LIN {X 0,Y 682.383,Z 707.31,A -85,B 0,C 180,E1 4367.128,E2 4367.128} C_VEL
LIN {X 0,Y 682.576,Z 707.31,A -85,B 0,C 180,E1 4371.565,E2 4371.565} C_VEL
LIN {X 0,Y 682.448,Z 707.31,A -85,B 0,C 180,E1 4374.859,E2 4374.859} C_VEL
LIN {X 0,Y 694.724,Z 736.712,A -85,B 0,C 180,E1 4375.905,E2 4375.905} C_VEL
LIN {X 0,Y 693.686,Z 780.447,A -85,B 0,C 180,E1 4376.761,E2 4376.761} C_VEL
LIN {X 0,Y 692.089,Z 825.553,A -85,B 0,C 180,E1 4378.187,E2 4378.187} C_VEL
LIN {X 0,Y 690.132,Z 869.734,A -85,B 0,C 180,E1 4380.196,E2 4380.196} C_VEL
LIN {X 0,Y 688.071,Z 912.153,A -85,B 0,C 180,E1 4382.814,E2 4382.814} C_VEL
LIN {X 0,Y 686.387,Z 948.211,A -85,B 0,C 180,E1 4385.72,E2 4385.72} C_VEL
LIN {X 0,Y 684.951,Z 981.072,A -85,B 0,C 180,E1 4389.145,E2 4389.145} C_VEL
LIN {X 0,Y 684.052,Z 1007.657,A -85,B 0,C 180,E1 4392.773,E2 4392.773} C_VEL
LIN {X 0,Y 683.489,Z 1028.052,A -85,B 0,C 180,E1 4396.539,E2 4396.539} C_VEL
LIN {X 0,Y 683.179,Z 1041.813,A -85,B 0,C 180,E1 4400.192,E2 4400.192} C_VEL
LIN {X 0,Y 683.173,Z 1049.91,A -85,B 0,C 180,E1 4403.633,E2 4403.633} C_VEL
LIN {X 0,Y 683.009,Z 1053.376,A -85,B 0,C 180,E1 4407.457,E2 4407.457} C_VEL
LIN {X 0,Y 683.089,Z 1051.321,A -85,B 0,C 180,E1 4411.272,E2 4411.272} C_VEL
LIN {X 0,Y 683.176,Z 1045.315,A -85,B 0,C 180,E1 4414.453,E2 4414.453} C_VEL
LIN {X 0,Y 683.301,Z 1034.031,A -85,B 0,C 180,E1 4417.968,E2 4417.968} C_VEL
LIN {X 0,Y 683.712,Z 1015.525,A -85,B 0,C 180,E1 4421.831,E2 4421.831} C_VEL
LIN {X 0,Y 684.513,Z 990.501,A -85,B 0,C 180,E1 4425.594,E2 4425.594} C_VEL
LIN {X 0,Y 685.858,Z 958.739,A -85,B 0,C 180,E1 4429.188,E2 4429.188} C_VEL
LIN {X 0,Y 687.532,Z 923.074,A -85,B 0,C 180,E1 4432.291,E2 4432.291} C_VEL
LIN {X 0,Y 689.545,Z 882.981,A -85,B 0,C 180,E1 4434.973,E2 4434.973} C_VEL
LIN {X 0,Y 691.593,Z 838.894,A -85,B 0,C 180,E1 4437.183,E2 4437.183} C_VEL
LIN {X 0,Y 693.261,Z 795.202,A -85,B 0,C 180,E1 4438.745,E2 4438.745} C_VEL
LIN {X 0,Y 694.501,Z 752.579,A -85,B 0,C 180,E1 4439.746,E2 4439.746} C_VEL
LIN {X 0,Y 693.995,Z 732.964,A -85,B 0,C 180,E1 4440.096,E2 4440.096} C_VEL
LIN {X 0,Y 682.507,Z 707.31,A -85,B 0,C 180,E1 4441.104,E2 4441.104} C_VEL
LIN {X 0,Y 682.451,Z 707.31,A -85,B 0,C 180,E1 4446.925,E2 4446.925} C_VEL
LIN {X 0,Y 682.413,Z 707.31,A -85,B 0,C 180,E1 4451.775,E2 4451.775} C_VEL
LIN {X 0,Y 682.5,Z 707.31,A -85,B 0,C 180,E1 4457.116,E2 4457.116} C_VEL
LIN {X 0,Y 682.473,Z 707.31,A -85,B 0,C 180,E1 4461.555,E2 4461.555} C_VEL
LIN {X 0,Y 682.507,Z 707.31,A -85,B 0,C 180,E1 4466.281,E2 4466.281} C_VEL
LIN {X 0,Y 682.478,Z 707.31,A -85,B 0,C 180,E1 4470.756,E2 4470.756} C_VEL
LIN {X 0,Y 682.492,Z 707.31,A -85,B 0,C 180,E1 4475.557,E2 4475.557} C_VEL
LIN {X 0,Y 682.591,Z 707.31,A -85,B 0,C 180,E1 4480.546,E2 4480.546} C_VEL
LIN {X 0,Y 682.835,Z 707.31,A -85,B 0,C 180,E1 4485.868,E2 4485.868} C_VEL
LIN {X 0,Y 682.918,Z 707.31,A -85,B 0,C 180,E1 4491.062,E2 4491.062} C_VEL
LIN {X 0,Y 682.761,Z 707.31,A -85,B 0,C 180,E1 4496.18,E2 4496.18} C_VEL
LIN {X 0,Y 683.022,Z 707.31,A -85,B 0,C 180,E1 4501.269,E2 4501.269} C_VEL
LIN {X 0,Y 682.964,Z 707.31,A -85,B 0,C 180,E1 4507.648,E2 4507.648} C_VEL
LIN {X 0,Y 682.688,Z 707.31,A -85,B 0,C 180,E1 4512.823,E2 4512.823} C_VEL
LIN {X 0,Y 682.453,Z 707.31,A -85,B 0,C 180,E1 4518.109,E2 4518.109} C_VEL
LIN {X 0,Y 682.435,Z 707.31,A -85,B 0,C 180,E1 4521.572,E2 4521.572} C_VEL
LIN {X 0,Y 678.414,Z 707.31,A -85,B 0,C 180,E1 4523.005,E2 4523.005} C_VEL
LIN {X 0,Y 674.479,Z 707.31,A -85,B 0,C 180,E1 4524.456,E2 4524.456} C_VEL
LIN {X 0,Y 674.601,Z 707.31,A -85,B 0,C 180,E1 4529.614,E2 4529.614} C_VEL
LIN {X 0,Y 674.601,Z 707.31,A -85,B 0,C 180,E1 4534.163,E2 4534.163} C_VEL
LIN {X 0,Y 674.578,Z 707.31,A -85,B 0,C 180,E1 4538.973,E2 4538.973} C_VEL
LIN {X 0,Y 674.535,Z 707.31,A -85,B 0,C 180,E1 4544.138,E2 4544.138} C_VEL
LIN {X 0,Y 674.52,Z 707.31,A -85,B 0,C 180,E1 4549.801,E2 4549.801} C_VEL
LIN {X 0,Y 674.478,Z 707.31,A -85,B 0,C 180,E1 4554.256,E2 4554.256} C_VEL
LIN {X 0,Y 674.508,Z 708.066,A -85,B 0,C 180,E1 4556.111,E2 4556.111} C_VEL
LIN {X 0,Y 688.176,Z 737.551,A -85,B 0,C 180,E1 4557.231,E2 4557.231} C_VEL
LIN {X 0,Y 687.447,Z 791.806,A -85,B 0,C 180,E1 4558.03,E2 4558.03} C_VEL
LIN {X 0,Y 685.87,Z 838.816,A -85,B 0,C 180,E1 4559.294,E2 4559.294} C_VEL
LIN {X 0,Y 683.746,Z 884.753,A -85,B 0,C 180,E1 4561.162,E2 4561.162} C_VEL
LIN {X 0,Y 681.479,Z 927.902,A -85,B 0,C 180,E1 4563.593,E2 4563.593} C_VEL
LIN {X 0,Y 679.459,Z 966.912,A -85,B 0,C 180,E1 4566.505,E2 4566.505} C_VEL
LIN {X 0,Y 677.682,Z 1000.895,A -85,B 0,C 180,E1 4569.793,E2 4569.793} C_VEL
LIN {X 0,Y 676.498,Z 1029.549,A -85,B 0,C 180,E1 4573.404,E2 4573.404} C_VEL
LIN {X 0,Y 675.771,Z 1053.159,A -85,B 0,C 180,E1 4577.409,E2 4577.409} C_VEL
LIN {X 0,Y 675.4,Z 1069.16,A -85,B 0,C 180,E1 4581.288,E2 4581.288} C_VEL
LIN {X 0,Y 675.235,Z 1078.459,A -85,B 0,C 180,E1 4584.849,E2 4584.849} C_VEL
LIN {X 0,Y 675.177,Z 1083.168,A -85,B 0,C 180,E1 4588.713,E2 4588.713} C_VEL
LIN {X 0,Y 675.3,Z 1082.218,A -85,B 0,C 180,E1 4592.572,E2 4592.572} C_VEL
LIN {X 0,Y 675.237,Z 1075.636,A -85,B 0,C 180,E1 4596.442,E2 4596.442} C_VEL
LIN {X 0,Y 675.368,Z 1064.65,A -85,B 0,C 180,E1 4599.981,E2 4599.981} C_VEL
LIN {X 0,Y 675.764,Z 1047.785,A -85,B 0,C 180,E1 4603.618,E2 4603.618} C_VEL
LIN {X 0,Y 676.601,Z 1025.27,A -85,B 0,C 180,E1 4607.192,E2 4607.192} C_VEL
LIN {X 0,Y 677.818,Z 997.464,A -85,B 0,C 180,E1 4610.573,E2 4610.573} C_VEL
LIN {X 0,Y 679.494,Z 964.868,A -85,B 0,C 180,E1 4613.667,E2 4613.667} C_VEL
LIN {X 0,Y 681.608,Z 926.092,A -85,B 0,C 180,E1 4616.52,E2 4616.52} C_VEL
LIN {X 0,Y 683.832,Z 883.698,A -85,B 0,C 180,E1 4618.886,E2 4618.886} C_VEL
LIN {X 0,Y 685.911,Z 837.811,A -85,B 0,C 180,E1 4620.74,E2 4620.74} C_VEL
LIN {X 0,Y 687.491,Z 790.369,A -85,B 0,C 180,E1 4622.002,E2 4622.002} C_VEL
LIN {X 0,Y 687.505,Z 735.67,A -85,B 0,C 180,E1 4622.828,E2 4622.828} C_VEL
LIN {X 0,Y 674.593,Z 707.31,A -85,B 0,C 180,E1 4623.954,E2 4623.954} C_VEL
LIN {X 0,Y 674.584,Z 707.31,A -85,B 0,C 180,E1 4628.975,E2 4628.975} C_VEL
LIN {X 0,Y 674.547,Z 707.31,A -85,B 0,C 180,E1 4634.14,E2 4634.14} C_VEL
LIN {X 0,Y 674.52,Z 707.31,A -85,B 0,C 180,E1 4639.804,E2 4639.804} C_VEL
LIN {X 0,Y 674.531,Z 707.31,A -85,B 0,C 180,E1 4644.263,E2 4644.263} C_VEL
LIN {X 0,Y 674.635,Z 707.31,A -85,B 0,C 180,E1 4648.896,E2 4648.896} C_VEL
LIN {X 0,Y 674.568,Z 707.31,A -85,B 0,C 180,E1 4654.736,E2 4654.736} C_VEL
LIN {X 0,Y 674.678,Z 707.31,A -85,B 0,C 180,E1 4660.623,E2 4660.623} C_VEL
LIN {X 0,Y 674.746,Z 707.31,A -85,B 0,C 180,E1 4665.7,E2 4665.7} C_VEL
LIN {X 0,Y 674.975,Z 707.31,A -85,B 0,C 180,E1 4671.056,E2 4671.056} C_VEL
LIN {X 0,Y 674.685,Z 707.31,A -85,B 0,C 180,E1 4674.848,E2 4674.848} C_VEL
LIN {X 0,Y 674.832,Z 707.31,A -85,B 0,C 180,E1 4680.002,E2 4680.002} C_VEL
LIN {X 0,Y 674.973,Z 707.31,A -85,B 0,C 180,E1 4685.155,E2 4685.155} C_VEL
LIN {X 0,Y 674.842,Z 707.31,A -85,B 0,C 180,E1 4691.662,E2 4691.662} C_VEL
LIN {X 0,Y 674.512,Z 707.31,A -85,B 0,C 180,E1 4696.984,E2 4696.984} C_VEL
LIN {X 0,Y 674.815,Z 707.31,A -85,B 0,C 180,E1 4701.06,E2 4701.06} C_VEL
LIN {X 0,Y 674.524,Z 707.31,A -85,B 0,C 180,E1 4706.021,E2 4706.021} C_VEL
LIN {X 0,Y 674.373,Z 707.31,A -85,B 0,C 180,E1 4711.362,E2 4711.362} C_VEL
LIN {X 0,Y 674.46,Z 707.31,A -85,B 0,C 180,E1 4716.016,E2 4716.016} C_VEL
LIN {X 0,Y 674.591,Z 707.31,A -85,B 0,C 180,E1 4720.654,E2 4720.654} C_VEL
LIN {X 0,Y 674.533,Z 707.31,A -85,B 0,C 180,E1 4725.967,E2 4725.967} C_VEL
LIN {X 0,Y 674.655,Z 707.31,A -85,B 0,C 180,E1 4731.831,E2 4731.831} C_VEL
LIN {X 0,Y 674.543,Z 707.726,A -85,B 0,C 180,E1 4734.439,E2 4734.439} C_VEL
LIN {X 0,Y 688.006,Z 738.757,A -85,B 0,C 180,E1 4735.584,E2 4735.584} C_VEL
LIN {X 0,Y 686.802,Z 782.385,A -85,B 0,C 180,E1 4736.467,E2 4736.467} C_VEL
LIN {X 0,Y 685.108,Z 826.206,A -85,B 0,C 180,E1 4737.881,E2 4737.881} C_VEL
LIN {X 0,Y 682.962,Z 870.549,A -85,B 0,C 180,E1 4739.927,E2 4739.927} C_VEL
LIN {X 0,Y 680.722,Z 912.029,A -85,B 0,C 180,E1 4742.514,E2 4742.514} C_VEL
LIN {X 0,Y 678.777,Z 949.734,A -85,B 0,C 180,E1 4745.606,E2 4745.606} C_VEL
LIN {X 0,Y 677.211,Z 981.864,A -85,B 0,C 180,E1 4749.021,E2 4749.021} C_VEL
LIN {X 0,Y 676.257,Z 1007.816,A -85,B 0,C 180,E1 4752.619,E2 4752.619} C_VEL
LIN {X 0,Y 675.644,Z 1027.935,A -85,B 0,C 180,E1 4756.379,E2 4756.379} C_VEL
LIN {X 0,Y 675.323,Z 1041.566,A -85,B 0,C 180,E1 4760.018,E2 4760.018} C_VEL
LIN {X 0,Y 675.273,Z 1049.865,A -85,B 0,C 180,E1 4763.558,E2 4763.558} C_VEL
LIN {X 0,Y 675.125,Z 1053.369,A -85,B 0,C 180,E1 4767.428,E2 4767.428} C_VEL
LIN {X 0,Y 675.205,Z 1051.353,A -85,B 0,C 180,E1 4771.287,E2 4771.287} C_VEL
LIN {X 0,Y 675.249,Z 1043.77,A -85,B 0,C 180,E1 4775.151,E2 4775.151} C_VEL
LIN {X 0,Y 675.418,Z 1031.467,A -85,B 0,C 180,E1 4778.711,E2 4778.711} C_VEL
LIN {X 0,Y 675.912,Z 1014.099,A -85,B 0,C 180,E1 4782.237,E2 4782.237} C_VEL
LIN {X 0,Y 676.833,Z 989.858,A -85,B 0,C 180,E1 4785.886,E2 4785.886} C_VEL
LIN {X 0,Y 678.252,Z 959.002,A -85,B 0,C 180,E1 4789.412,E2 4789.412} C_VEL
LIN {X 0,Y 680.132,Z 922.968,A -85,B 0,C 180,E1 4792.581,E2 4792.581} C_VEL
LIN {X 0,Y 682.333,Z 883.236,A -85,B 0,C 180,E1 4795.267,E2 4795.267} C_VEL
LIN {X 0,Y 684.626,Z 838.791,A -85,B 0,C 180,E1 4797.514,E2 4797.514} C_VEL
LIN {X 0,Y 686.388,Z 796.028,A -85,B 0,C 180,E1 4799.06,E2 4799.06} C_VEL
LIN {X 0,Y 687.752,Z 754.022,A -85,B 0,C 180,E1 4800.068,E2 4800.068} C_VEL
LIN {X 0,Y 687.42,Z 735.913,A -85,B 0,C 180,E1 4800.398,E2 4800.398} C_VEL
LIN {X 0,Y 674.524,Z 707.31,A -85,B 0,C 180,E1 4801.552,E2 4801.552} C_VEL
LIN {X 0,Y 674.521,Z 707.31,A -85,B 0,C 180,E1 4807.344,E2 4807.344} C_VEL
LIN {X 0,Y 674.469,Z 707.31,A -85,B 0,C 180,E1 4812.38,E2 4812.38} C_VEL
LIN {X 0,Y 674.605,Z 707.31,A -85,B 0,C 180,E1 4817.843,E2 4817.843} C_VEL
LIN {X 0,Y 674.527,Z 707.31,A -85,B 0,C 180,E1 4822.655,E2 4822.655} C_VEL
LIN {X 0,Y 674.622,Z 707.31,A -85,B 0,C 180,E1 4827.375,E2 4827.375} C_VEL
LIN {X 0,Y 674.57,Z 707.31,A -85,B 0,C 180,E1 4831.849,E2 4831.849} C_VEL
LIN {X 0,Y 674.476,Z 707.31,A -85,B 0,C 180,E1 4837.101,E2 4837.101} C_VEL
LIN {X 0,Y 674.536,Z 707.31,A -85,B 0,C 180,E1 4841.666,E2 4841.666} C_VEL
LIN {X 0,Y 675.041,Z 707.31,A -85,B 0,C 180,E1 4847.025,E2 4847.025} C_VEL
LIN {X 0,Y 674.947,Z 707.31,A -85,B 0,C 180,E1 4852.256,E2 4852.256} C_VEL
LIN {X 0,Y 674.865,Z 707.31,A -85,B 0,C 180,E1 4856.135,E2 4856.135} C_VEL
LIN {X 0,Y 675.128,Z 707.31,A -85,B 0,C 180,E1 4861.284,E2 4861.284} C_VEL
LIN {X 0,Y 675.046,Z 707.31,A -85,B 0,C 180,E1 4867.738,E2 4867.738} C_VEL
LIN {X 0,Y 674.77,Z 707.31,A -85,B 0,C 180,E1 4872.976,E2 4872.976} C_VEL
LIN {X 0,Y 674.551,Z 707.31,A -85,B 0,C 180,E1 4878.329,E2 4878.329} C_VEL
LIN {X 0,Y 674.451,Z 707.31,A -85,B 0,C 180,E1 4882.894,E2 4882.894} C_VEL
LIN {X 0,Y 674.479,Z 707.31,A -85,B 0,C 180,E1 4884.456,E2 4884.456} C_VEL
LIN {X 0,Y 670.595,Z 707.31,A -85,B 0,C 180,E1 4885.904,E2 4885.904} C_VEL
LIN {X 0,Y 666.66,Z 707.31,A -85,B 0,C 180,E1 4887.369,E2 4887.369} C_VEL
LIN {X 0,Y 666.712,Z 707.31,A -85,B 0,C 180,E1 4893.056,E2 4893.056} C_VEL
LIN {X 0,Y 666.637,Z 707.31,A -85,B 0,C 180,E1 4897.859,E2 4897.859} C_VEL
LIN {X 0,Y 666.548,Z 707.31,A -85,B 0,C 180,E1 4903.32,E2 4903.32} C_VEL
LIN {X 0,Y 666.538,Z 707.31,A -85,B 0,C 180,E1 4908.751,E2 4908.751} C_VEL
LIN {X 0,Y 666.576,Z 707.31,A -85,B 0,C 180,E1 4913.765,E2 4913.765} C_VEL
LIN {X 0,Y 666.565,Z 707.31,A -85,B 0,C 180,E1 4915.64,E2 4915.64} C_VEL
LIN {X 0,Y 681.528,Z 740.134,A -85,B 0,C 180,E1 4916.902,E2 4916.902} C_VEL
LIN {X 0,Y 680.677,Z 792.992,A -85,B 0,C 180,E1 4917.702,E2 4917.702} C_VEL
LIN {X 0,Y 678.976,Z 839.749,A -85,B 0,C 180,E1 4918.984,E2 4918.984} C_VEL
LIN {X 0,Y 676.703,Z 884.982,A -85,B 0,C 180,E1 4920.845,E2 4920.845} C_VEL
LIN {X 0,Y 674.264,Z 927.901,A -85,B 0,C 180,E1 4923.288,E2 4923.288} C_VEL
LIN {X 0,Y 671.967,Z 966.911,A -85,B 0,C 180,E1 4926.227,E2 4926.227} C_VEL
LIN {X 0,Y 670.1,Z 1000.051,A -85,B 0,C 180,E1 4929.459,E2 4929.459} C_VEL
LIN {X 0,Y 668.709,Z 1029.55,A -85,B 0,C 180,E1 4933.205,E2 4933.205} C_VEL
LIN {X 0,Y 667.954,Z 1052.672,A -85,B 0,C 180,E1 4937.157,E2 4937.157} C_VEL
LIN {X 0,Y 667.533,Z 1069.16,A -85,B 0,C 180,E1 4941.185,E2 4941.185} C_VEL
LIN {X 0,Y 667.352,Z 1078.459,A -85,B 0,C 180,E1 4944.788,E2 4944.788} C_VEL
LIN {X 0,Y 667.278,Z 1083.167,A -85,B 0,C 180,E1 4948.698,E2 4948.698} C_VEL
LIN {X 0,Y 667.428,Z 1082.217,A -85,B 0,C 180,E1 4952.602,E2 4952.602} C_VEL
LIN {X 0,Y 667.344,Z 1075.636,A -85,B 0,C 180,E1 4956.519,E2 4956.519} C_VEL
LIN {X 0,Y 667.512,Z 1064.516,A -85,B 0,C 180,E1 4960.133,E2 4960.133} C_VEL
LIN {X 0,Y 668.06,Z 1046.033,A -85,B 0,C 180,E1 4964.113,E2 4964.113} C_VEL
LIN {X 0,Y 669.136,Z 1021.013,A -85,B 0,C 180,E1 4967.987,E2 4967.987} C_VEL
LIN {X 0,Y 670.698,Z 989.205,A -85,B 0,C 180,E1 4971.691,E2 4971.691} C_VEL
LIN {X 0,Y 672.742,Z 953.245,A -85,B 0,C 180,E1 4974.894,E2 4974.894} C_VEL
LIN {X 0,Y 675.122,Z 912.935,A -85,B 0,C 180,E1 4977.647,E2 4977.647} C_VEL
LIN {X 0,Y 677.594,Z 868.414,A -85,B 0,C 180,E1 4979.913,E2 4979.913} C_VEL
LIN {X 0,Y 679.642,Z 822.708,A -85,B 0,C 180,E1 4981.559,E2 4981.559} C_VEL
LIN {X 0,Y 681.145,Z 773.641,A -85,B 0,C 180,E1 4982.662,E2 4982.662} C_VEL
LIN {X 0,Y 680.831,Z 737.977,A -85,B 0,C 180,E1 4983.163,E2 4983.163} C_VEL
LIN {X 0,Y 666.664,Z 707.31,A -85,B 0,C 180,E1 4984.388,E2 4984.388} C_VEL
LIN {X 0,Y 666.651,Z 707.31,A -85,B 0,C 180,E1 4989.529,E2 4989.529} C_VEL
LIN {X 0,Y 666.561,Z 707.31,A -85,B 0,C 180,E1 4995.193,E2 4995.193} C_VEL
LIN {X 0,Y 666.634,Z 707.31,A -85,B 0,C 180,E1 5000.613,E2 5000.613} C_VEL
LIN {X 0,Y 666.621,Z 707.31,A -85,B 0,C 180,E1 5005.371,E2 5005.371} C_VEL
LIN {X 0,Y 666.665,Z 707.31,A -85,B 0,C 180,E1 5009.998,E2 5009.998} C_VEL
LIN {X 0,Y 666.584,Z 707.31,A -85,B 0,C 180,E1 5015.414,E2 5015.414} C_VEL
LIN {X 0,Y 666.727,Z 707.31,A -85,B 0,C 180,E1 5020.069,E2 5020.069} C_VEL
LIN {X 0,Y 666.82,Z 707.31,A -85,B 0,C 180,E1 5025.526,E2 5025.526} C_VEL
LIN {X 0,Y 667.069,Z 707.31,A -85,B 0,C 180,E1 5030.852,E2 5030.852} C_VEL
LIN {X 0,Y 666.809,Z 707.31,A -85,B 0,C 180,E1 5034.787,E2 5034.787} C_VEL
LIN {X 0,Y 666.943,Z 707.31,A -85,B 0,C 180,E1 5040.002,E2 5040.002} C_VEL
LIN {X 0,Y 667.051,Z 707.31,A -85,B 0,C 180,E1 5045.216,E2 5045.216} C_VEL
LIN {X 0,Y 666.911,Z 707.31,A -85,B 0,C 180,E1 5051.803,E2 5051.803} C_VEL
LIN {X 0,Y 666.589,Z 707.31,A -85,B 0,C 180,E1 5057.292,E2 5057.292} C_VEL
LIN {X 0,Y 666.887,Z 707.31,A -85,B 0,C 180,E1 5061.322,E2 5061.322} C_VEL
LIN {X 0,Y 666.657,Z 707.31,A -85,B 0,C 180,E1 5065.59,E2 5065.59} C_VEL
LIN {X 0,Y 666.486,Z 707.31,A -85,B 0,C 180,E1 5070.231,E2 5070.231} C_VEL
LIN {X 0,Y 666.516,Z 707.31,A -85,B 0,C 180,E1 5075.066,E2 5075.066} C_VEL
LIN {X 0,Y 666.674,Z 707.31,A -85,B 0,C 180,E1 5079.531,E2 5079.531} C_VEL
LIN {X 0,Y 666.582,Z 707.31,A -85,B 0,C 180,E1 5085.192,E2 5085.192} C_VEL
LIN {X 0,Y 666.718,Z 707.31,A -85,B 0,C 180,E1 5090.608,E2 5090.608} C_VEL
LIN {X 0,Y 666.656,Z 707.711,A -85,B 0,C 180,E1 5093.986,E2 5093.986} C_VEL
LIN {X 0,Y 681.297,Z 740.305,A -85,B 0,C 180,E1 5095.248,E2 5095.248} C_VEL
LIN {X 0,Y 679.935,Z 785.032,A -85,B 0,C 180,E1 5096.188,E2 5096.188} C_VEL
LIN {X 0,Y 678.07,Z 828.293,A -85,B 0,C 180,E1 5097.627,E2 5097.627} C_VEL
LIN {X 0,Y 675.759,Z 871.521,A -85,B 0,C 180,E1 5099.659,E2 5099.659} C_VEL
LIN {X 0,Y 673.373,Z 912.455,A -85,B 0,C 180,E1 5102.25,E2 5102.25} C_VEL
LIN {X 0,Y 671.228,Z 949.46,A -85,B 0,C 180,E1 5105.313,E2 5105.313} C_VEL
LIN {X 0,Y 669.5,Z 981.657,A -85,B 0,C 180,E1 5108.768,E2 5108.768} C_VEL
LIN {X 0,Y 668.432,Z 1008.425,A -85,B 0,C 180,E1 5112.537,E2 5112.537} C_VEL
LIN {X 0,Y 667.727,Z 1029.34,A -85,B 0,C 180,E1 5116.549,E2 5116.549} C_VEL
LIN {X 0,Y 667.406,Z 1042.365,A -85,B 0,C 180,E1 5120.196,E2 5120.196} C_VEL
LIN {X 0,Y 667.373,Z 1049.821,A -85,B 0,C 180,E1 5123.482,E2 5123.482} C_VEL
LIN {X 0,Y 667.228,Z 1053.363,A -85,B 0,C 180,E1 5127.397,E2 5127.397} C_VEL
LIN {X 0,Y 667.304,Z 1051.385,A -85,B 0,C 180,E1 5131.302,E2 5131.302} C_VEL
LIN {X 0,Y 667.367,Z 1043.842,A -85,B 0,C 180,E1 5135.212,E2 5135.212} C_VEL
LIN {X 0,Y 667.552,Z 1031.573,A -85,B 0,C 180,E1 5138.814,E2 5138.814} C_VEL
LIN {X 0,Y 668.097,Z 1013.892,A -85,B 0,C 180,E1 5142.443,E2 5142.443} C_VEL
LIN {X 0,Y 669.101,Z 989.793,A -85,B 0,C 180,E1 5146.108,E2 5146.108} C_VEL
LIN {X 0,Y 670.644,Z 959.267,A -85,B 0,C 180,E1 5149.641,E2 5149.641} C_VEL
LIN {X 0,Y 672.762,Z 923.021,A -85,B 0,C 180,E1 5152.865,E2 5152.865} C_VEL
LIN {X 0,Y 675.23,Z 882.54,A -85,B 0,C 180,E1 5155.621,E2 5155.621} C_VEL
LIN {X 0,Y 677.681,Z 838.342,A -85,B 0,C 180,E1 5157.867,E2 5157.867} C_VEL
LIN {X 0,Y 679.638,Z 794.078,A -85,B 0,C 180,E1 5159.469,E2 5159.469} C_VEL
LIN {X 0,Y 681.118,Z 751.141,A -85,B 0,C 180,E1 5160.474,E2 5160.474} C_VEL
LIN {X 0,Y 680.665,Z 738.196,A -85,B 0,C 180,E1 5160.727,E2 5160.727} C_VEL
LIN {X 0,Y 666.588,Z 707.31,A -85,B 0,C 180,E1 5161.955,E2 5161.955} C_VEL
LIN {X 0,Y 666.639,Z 707.31,A -85,B 0,C 180,E1 5167.863,E2 5167.863} C_VEL
LIN {X 0,Y 666.541,Z 707.31,A -85,B 0,C 180,E1 5173.318,E2 5173.318} C_VEL
LIN {X 0,Y 666.647,Z 707.31,A -85,B 0,C 180,E1 5178.757,E2 5178.757} C_VEL
LIN {X 0,Y 666.62,Z 707.31,A -85,B 0,C 180,E1 5183.766,E2 5183.766} C_VEL
LIN {X 0,Y 666.726,Z 707.31,A -85,B 0,C 180,E1 5188.48,E2 5188.48} C_VEL
LIN {X 0,Y 666.702,Z 707.31,A -85,B 0,C 180,E1 5194.412,E2 5194.412} C_VEL
LIN {X 0,Y 666.74,Z 707.31,A -85,B 0,C 180,E1 5200.064,E2 5200.064} C_VEL
LIN {X 0,Y 666.936,Z 707.31,A -85,B 0,C 180,E1 5205.524,E2 5205.524} C_VEL
LIN {X 0,Y 667.092,Z 707.31,A -85,B 0,C 180,E1 5210.848,E2 5210.848} C_VEL
LIN {X 0,Y 666.985,Z 707.31,A -85,B 0,C 180,E1 5216.089,E2 5216.089} C_VEL
LIN {X 0,Y 667.058,Z 707.31,A -85,B 0,C 180,E1 5221.648,E2 5221.648} C_VEL
LIN {X 0,Y 667.131,Z 707.31,A -85,B 0,C 180,E1 5227.831,E2 5227.831} C_VEL
LIN {X 0,Y 666.862,Z 707.31,A -85,B 0,C 180,E1 5233.132,E2 5233.132} C_VEL
LIN {X 0,Y 666.661,Z 707.31,A -85,B 0,C 180,E1 5238.554,E2 5238.554} C_VEL
LIN {X 0,Y 666.562,Z 707.31,A -85,B 0,C 180,E1 5242.733,E2 5242.733} C_VEL
LIN {X 0,Y 666.66,Z 707.31,A -85,B 0,C 180,E1 5247.369,E2 5247.369} C_VEL
LIN {X 0,Y 662.663,Z 707.31,A -85,B 0,C 180,E1 5248.838,E2 5248.838} C_VEL
LIN {X 0,Y 658.79,Z 707.31,A -85,B 0,C 180,E1 5250.325,E2 5250.325} C_VEL
LIN {X 0,Y 658.748,Z 707.31,A -85,B 0,C 180,E1 5255.104,E2 5255.104} C_VEL
LIN {X 0,Y 658.617,Z 707.31,A -85,B 0,C 180,E1 5260.597,E2 5260.597} C_VEL
LIN {X 0,Y 658.605,Z 707.31,A -85,B 0,C 180,E1 5266.347,E2 5266.347} C_VEL
LIN {X 0,Y 658.665,Z 707.31,A -85,B 0,C 180,E1 5271.596,E2 5271.596} C_VEL
LIN {X 0,Y 658.652,Z 707.31,A -85,B 0,C 180,E1 5275.154,E2 5275.154} C_VEL
LIN {X 0,Y 674.979,Z 744.406,A -85,B 0,C 180,E1 5276.592,E2 5276.592} C_VEL
LIN {X 0,Y 673.878,Z 795.428,A -85,B 0,C 180,E1 5277.395,E2 5277.395} C_VEL
LIN {X 0,Y 672.06,Z 841.218,A -85,B 0,C 180,E1 5278.686,E2 5278.686} C_VEL
LIN {X 0,Y 669.655,Z 885.266,A -85,B 0,C 180,E1 5280.524,E2 5280.524} C_VEL
LIN {X 0,Y 667.052,Z 927.898,A -85,B 0,C 180,E1 5282.976,E2 5282.976} C_VEL
LIN {X 0,Y 664.557,Z 966.671,A -85,B 0,C 180,E1 5285.923,E2 5285.923} C_VEL
LIN {X 0,Y 662.406,Z 1001.472,A -85,B 0,C 180,E1 5289.375,E2 5289.375} C_VEL
LIN {X 0,Y 660.916,Z 1029.551,A -85,B 0,C 180,E1 5293.001,E2 5293.001} C_VEL
LIN {X 0,Y 660.098,Z 1052.401,A -85,B 0,C 180,E1 5296.948,E2 5296.948} C_VEL
LIN {X 0,Y 659.682,Z 1068.937,A -85,B 0,C 180,E1 5301.014,E2 5301.014} C_VEL
LIN {X 0,Y 659.459,Z 1078.458,A -85,B 0,C 180,E1 5304.725,E2 5304.725} C_VEL
LIN {X 0,Y 659.395,Z 1083.167,A -85,B 0,C 180,E1 5308.683,E2 5308.683} C_VEL
LIN {X 0,Y 659.526,Z 1082.217,A -85,B 0,C 180,E1 5312.633,E2 5312.633} C_VEL
LIN {X 0,Y 659.452,Z 1075.636,A -85,B 0,C 180,E1 5316.597,E2 5316.597} C_VEL
LIN {X 0,Y 659.711,Z 1063.177,A -85,B 0,C 180,E1 5320.589,E2 5320.589} C_VEL
LIN {X 0,Y 660.247,Z 1046.034,A -85,B 0,C 180,E1 5324.284,E2 5324.284} C_VEL
LIN {X 0,Y 661.397,Z 1021.015,A -85,B 0,C 180,E1 5328.205,E2 5328.205} C_VEL
LIN {X 0,Y 663.093,Z 989.816,A -85,B 0,C 180,E1 5331.889,E2 5331.889} C_VEL
LIN {X 0,Y 665.395,Z 953.247,A -85,B 0,C 180,E1 5335.188,E2 5335.188} C_VEL
LIN {X 0,Y 668.026,Z 912.349,A -85,B 0,C 180,E1 5338.002,E2 5338.002} C_VEL
LIN {X 0,Y 670.575,Z 869.78,A -85,B 0,C 180,E1 5340.196,E2 5340.196} C_VEL
LIN {X 0,Y 672.86,Z 822.907,A -85,B 0,C 180,E1 5341.908,E2 5341.908} C_VEL
LIN {X 0,Y 674.477,Z 773.631,A -85,B 0,C 180,E1 5343.026,E2 5343.026} C_VEL
LIN {X 0,Y 674.327,Z 740.95,A -85,B 0,C 180,E1 5343.487,E2 5343.487} C_VEL
LIN {X 0,Y 658.734,Z 707.31,A -85,B 0,C 180,E1 5344.851,E2 5344.851} C_VEL
LIN {X 0,Y 658.674,Z 707.31,A -85,B 0,C 180,E1 5350.609,E2 5350.609} C_VEL
LIN {X 0,Y 658.603,Z 707.31,A -85,B 0,C 180,E1 5356.352,E2 5356.352} C_VEL
LIN {X 0,Y 658.676,Z 707.31,A -85,B 0,C 180,E1 5361.601,E2 5361.601} C_VEL
LIN {X 0,Y 658.747,Z 707.31,A -85,B 0,C 180,E1 5366.492,E2 5366.492} C_VEL
LIN {X 0,Y 658.728,Z 707.31,A -85,B 0,C 180,E1 5371.115,E2 5371.115} C_VEL
LIN {X 0,Y 658.681,Z 707.31,A -85,B 0,C 180,E1 5375.539,E2 5375.539} C_VEL
LIN {X 0,Y 658.744,Z 707.31,A -85,B 0,C 180,E1 5381.215,E2 5381.215} C_VEL
LIN {X 0,Y 658.928,Z 707.31,A -85,B 0,C 180,E1 5386.707,E2 5386.707} C_VEL
LIN {X 0,Y 659.21,Z 707.31,A -85,B 0,C 180,E1 5392.075,E2 5392.075} C_VEL
LIN {X 0,Y 659.302,Z 707.31,A -85,B 0,C 180,E1 5398.685,E2 5398.685} C_VEL
LIN {X 0,Y 659.119,Z 707.31,A -85,B 0,C 180,E1 5405.279,E2 5405.279} C_VEL
LIN {X 0,Y 659.015,Z 707.31,A -85,B 0,C 180,E1 5410.603,E2 5410.603} C_VEL
LIN {X 0,Y 658.773,Z 707.31,A -85,B 0,C 180,E1 5416.026,E2 5416.026} C_VEL
LIN {X 0,Y 658.948,Z 707.31,A -85,B 0,C 180,E1 5421.592,E2 5421.592} C_VEL
LIN {X 0,Y 658.649,Z 707.31,A -85,B 0,C 180,E1 5426.196,E2 5426.196} C_VEL
LIN {X 0,Y 658.574,Z 707.31,A -85,B 0,C 180,E1 5431.956,E2 5431.956} C_VEL
LIN {X 0,Y 658.663,Z 707.31,A -85,B 0,C 180,E1 5436.743,E2 5436.743} C_VEL
LIN {X 0,Y 658.698,Z 707.31,A -85,B 0,C 180,E1 5441.852,E2 5441.852} C_VEL
LIN {X 0,Y 658.603,Z 707.31,A -85,B 0,C 180,E1 5447.42,E2 5447.42} C_VEL
LIN {X 0,Y 658.787,Z 707.31,A -85,B 0,C 180,E1 5451.606,E2 5451.606} C_VEL
LIN {X 0,Y 658.773,Z 707.954,A -85,B 0,C 180,E1 5453.523,E2 5453.523} C_VEL
LIN {X 0,Y 674.605,Z 743.976,A -85,B 0,C 180,E1 5454.943,E2 5454.943} C_VEL
LIN {X 0,Y 673.033,Z 789.763,A -85,B 0,C 180,E1 5455.96,E2 5455.96} C_VEL
LIN {X 0,Y 670.914,Z 833.503,A -85,B 0,C 180,E1 5457.497,E2 5457.497} C_VEL
LIN {X 0,Y 668.48,Z 874.159,A -85,B 0,C 180,E1 5459.481,E2 5459.481} C_VEL
LIN {X 0,Y 665.977,Z 913.837,A -85,B 0,C 180,E1 5462.052,E2 5462.052} C_VEL
LIN {X 0,Y 663.674,Z 949.184,A -85,B 0,C 180,E1 5465.013,E2 5465.013} C_VEL
LIN {X 0,Y 661.805,Z 981.45,A -85,B 0,C 180,E1 5468.509,E2 5468.509} C_VEL
LIN {X 0,Y 660.661,Z 1008.275,A -85,B 0,C 180,E1 5472.325,E2 5472.325} C_VEL
LIN {X 0,Y 659.899,Z 1029.234,A -85,B 0,C 180,E1 5476.386,E2 5476.386} C_VEL
LIN {X 0,Y 659.545,Z 1042.292,A -85,B 0,C 180,E1 5480.078,E2 5480.078} C_VEL
LIN {X 0,Y 659.474,Z 1049.776,A -85,B 0,C 180,E1 5483.403,E2 5483.403} C_VEL
LIN {X 0,Y 659.328,Z 1053.357,A -85,B 0,C 180,E1 5487.366,E2 5487.366} C_VEL
LIN {X 0,Y 659.422,Z 1051.417,A -85,B 0,C 180,E1 5491.317,E2 5491.317} C_VEL
LIN {X 0,Y 659.474,Z 1043.912,A -85,B 0,C 180,E1 5495.274,E2 5495.274} C_VEL
LIN {X 0,Y 659.713,Z 1031.462,A -85,B 0,C 180,E1 5498.972,E2 5498.972} C_VEL
LIN {X 0,Y 660.248,Z 1014.227,A -85,B 0,C 180,E1 5502.561,E2 5502.561} C_VEL
LIN {X 0,Y 661.401,Z 989.991,A -85,B 0,C 180,E1 5506.301,E2 5506.301} C_VEL
LIN {X 0,Y 663.082,Z 959.526,A -85,B 0,C 180,E1 5509.875,E2 5509.875} C_VEL
LIN {X 0,Y 665.371,Z 923.369,A -85,B 0,C 180,E1 5513.134,E2 5513.134} C_VEL
LIN {X 0,Y 668.075,Z 882.487,A -85,B 0,C 180,E1 5515.946,E2 5515.946} C_VEL
LIN {X 0,Y 670.724,Z 838.214,A -85,B 0,C 180,E1 5518.216,E2 5518.216} C_VEL
LIN {X 0,Y 672.86,Z 793.545,A -85,B 0,C 180,E1 5519.841,E2 5519.841} C_VEL
LIN {X 0,Y 674.506,Z 748.599,A -85,B 0,C 180,E1 5520.883,E2 5520.883} C_VEL
LIN {X 0,Y 673.551,Z 739.758,A -85,B 0,C 180,E1 5521.094,E2 5521.094} C_VEL
LIN {X 0,Y 658.678,Z 707.31,A -85,B 0,C 180,E1 5522.419,E2 5522.419} C_VEL
LIN {X 0,Y 658.697,Z 707.31,A -85,B 0,C 180,E1 5528.402,E2 5528.402} C_VEL
LIN {X 0,Y 658.642,Z 707.31,A -85,B 0,C 180,E1 5534.498,E2 5534.498} C_VEL
LIN {X 0,Y 658.706,Z 707.31,A -85,B 0,C 180,E1 5539.895,E2 5539.895} C_VEL
LIN {X 0,Y 658.722,Z 707.31,A -85,B 0,C 180,E1 5544.889,E2 5544.889} C_VEL
LIN {X 0,Y 658.783,Z 707.31,A -85,B 0,C 180,E1 5549.596,E2 5549.596} C_VEL
LIN {X 0,Y 658.763,Z 707.31,A -85,B 0,C 180,E1 5554.081,E2 5554.081} C_VEL
LIN {X 0,Y 658.809,Z 707.31,A -85,B 0,C 180,E1 5559.814,E2 5559.814} C_VEL
LIN {X 0,Y 658.984,Z 707.31,A -85,B 0,C 180,E1 5565.345,E2 5565.345} C_VEL
LIN {X 0,Y 659.187,Z 707.31,A -85,B 0,C 180,E1 5570.737,E2 5570.737} C_VEL
LIN {X 0,Y 659.086,Z 707.31,A -85,B 0,C 180,E1 5576.042,E2 5576.042} C_VEL
LIN {X 0,Y 659.321,Z 707.31,A -85,B 0,C 180,E1 5581.315,E2 5581.315} C_VEL
LIN {X 0,Y 659.216,Z 707.31,A -85,B 0,C 180,E1 5587.925,E2 5587.925} C_VEL
LIN {X 0,Y 658.939,Z 707.31,A -85,B 0,C 180,E1 5593.293,E2 5593.293} C_VEL
LIN {X 0,Y 658.747,Z 707.31,A -85,B 0,C 180,E1 5598.785,E2 5598.785} C_VEL
LIN {X 0,Y 658.69,Z 707.31,A -85,B 0,C 180,E1 5604.46,E2 5604.46} C_VEL
LIN {X 0,Y 658.748,Z 707.31,A -85,B 0,C 180,E1 5609.053,E2 5609.053} C_VEL
LIN {X 0,Y 658.79,Z 707.31,A -85,B 0,C 180,E1 5610.325,E2 5610.325} C_VEL
LIN {X 0,Y 654.875,Z 707.31,A -85,B 0,C 180,E1 5611.809,E2 5611.809} C_VEL
LIN {X 0,Y 650.798,Z 707.31,A -85,B 0,C 180,E1 5613.311,E2 5613.311} C_VEL
LIN {X 0,Y 650.728,Z 707.31,A -85,B 0,C 180,E1 5618.956,E2 5618.956} C_VEL
LIN {X 0,Y 650.723,Z 707.31,A -85,B 0,C 180,E1 5624.314,E2 5624.314} C_VEL
LIN {X 0,Y 650.71,Z 707.31,A -85,B 0,C 180,E1 5630.216,E2 5630.216} C_VEL
LIN {X 0,Y 650.771,Z 708.072,A -85,B 0,C 180,E1 5634.706,E2 5634.706} C_VEL
LIN {X 0,Y 668.221,Z 745.081,A -85,B 0,C 180,E1 5636.22,E2 5636.22} C_VEL
LIN {X 0,Y 667.2,Z 795.536,A -85,B 0,C 180,E1 5637.031,E2 5637.031} C_VEL
LIN {X 0,Y 665.398,Z 839.116,A -85,B 0,C 180,E1 5638.254,E2 5638.254} C_VEL
LIN {X 0,Y 662.786,Z 883.544,A -85,B 0,C 180,E1 5640.097,E2 5640.097} C_VEL
LIN {X 0,Y 659.923,Z 926.813,A -85,B 0,C 180,E1 5642.585,E2 5642.585} C_VEL
LIN {X 0,Y 657.123,Z 966.671,A -85,B 0,C 180,E1 5645.633,E2 5645.633} C_VEL
LIN {X 0,Y 654.879,Z 1000.243,A -85,B 0,C 180,E1 5648.981,E2 5648.981} C_VEL
LIN {X 0,Y 653.155,Z 1029.552,A -85,B 0,C 180,E1 5652.793,E2 5652.793} C_VEL
LIN {X 0,Y 652.277,Z 1052.472,A -85,B 0,C 180,E1 5656.803,E2 5656.803} C_VEL
LIN {X 0,Y 651.821,Z 1068.011,A -85,B 0,C 180,E1 5660.633,E2 5660.633} C_VEL
LIN {X 0,Y 651.669,Z 1077.194,A -85,B 0,C 180,E1 5663.993,E2 5663.993} C_VEL
LIN {X 0,Y 651.598,Z 1082.215,A -85,B 0,C 180,E1 5667.333,E2 5667.333} C_VEL
LIN {X 0,Y 651.669,Z 1083.167,A -85,B 0,C 180,E1 5671.332,E2 5671.332} C_VEL
LIN {X 0,Y 651.539,Z 1078.461,A -85,B 0,C 180,E1 5675.338,E2 5675.338} C_VEL
LIN {X 0,Y 651.669,Z 1069.728,A -85,B 0,C 180,E1 5678.864,E2 5678.864} C_VEL
LIN {X 0,Y 652.114,Z 1053.871,A -85,B 0,C 180,E1 5682.899,E2 5682.899} C_VEL
LIN {X 0,Y 652.913,Z 1032.85,A -85,B 0,C 180,E1 5686.691,E2 5686.691} C_VEL
LIN {X 0,Y 654.288,Z 1007.601,A -85,B 0,C 180,E1 5690.152,E2 5690.152} C_VEL
LIN {X 0,Y 656.365,Z 976.941,A -85,B 0,C 180,E1 5693.43,E2 5693.43} C_VEL
LIN {X 0,Y 659.024,Z 939.452,A -85,B 0,C 180,E1 5696.537,E2 5696.537} C_VEL
LIN {X 0,Y 661.881,Z 898.25,A -85,B 0,C 180,E1 5699.139,E2 5699.139} C_VEL
LIN {X 0,Y 664.589,Z 854.247,A -85,B 0,C 180,E1 5701.191,E2 5701.191} C_VEL
LIN {X 0,Y 666.78,Z 809.272,A -85,B 0,C 180,E1 5702.639,E2 5702.639} C_VEL
LIN {X 0,Y 668.057,Z 764.647,A -85,B 0,C 180,E1 5703.522,E2 5703.522} C_VEL
LIN {X 0,Y 667.491,Z 742.929,A -85,B 0,C 180,E1 5703.849,E2 5703.849} C_VEL
LIN {X 0,Y 650.834,Z 707.31,A -85,B 0,C 180,E1 5705.373,E2 5705.373} C_VEL
LIN {X 0,Y 650.774,Z 707.31,A -85,B 0,C 180,E1 5710.693,E2 5710.693} C_VEL
LIN {X 0,Y 650.711,Z 707.31,A -85,B 0,C 180,E1 5716.214,E2 5716.214} C_VEL
LIN {X 0,Y 650.715,Z 707.31,A -85,B 0,C 180,E1 5721.043,E2 5721.043} C_VEL
LIN {X 0,Y 650.818,Z 707.31,A -85,B 0,C 180,E1 5726.029,E2 5726.029} C_VEL
LIN {X 0,Y 650.83,Z 707.31,A -85,B 0,C 180,E1 5730.731,E2 5730.731} C_VEL
LIN {X 0,Y 650.778,Z 707.31,A -85,B 0,C 180,E1 5735.25,E2 5735.25} C_VEL
LIN {X 0,Y 650.846,Z 707.31,A -85,B 0,C 180,E1 5740.979,E2 5740.979} C_VEL
LIN {X 0,Y 651.013,Z 707.31,A -85,B 0,C 180,E1 5746.542,E2 5746.542} C_VEL
LIN {X 0,Y 651.325,Z 707.31,A -85,B 0,C 180,E1 5751.978,E2 5751.978} C_VEL
LIN {X 0,Y 651.419,Z 707.31,A -85,B 0,C 180,E1 5758.669,E2 5758.669} C_VEL
LIN {X 0,Y 651.196,Z 707.31,A -85,B 0,C 180,E1 5765.343,E2 5765.343} C_VEL
LIN {X 0,Y 651.098,Z 707.31,A -85,B 0,C 180,E1 5770.733,E2 5770.733} C_VEL
LIN {X 0,Y 650.839,Z 707.31,A -85,B 0,C 180,E1 5776.227,E2 5776.227} C_VEL
LIN {X 0,Y 651.016,Z 707.31,A -85,B 0,C 180,E1 5781.868,E2 5781.868} C_VEL
LIN {X 0,Y 650.769,Z 707.31,A -85,B 0,C 180,E1 5786.262,E2 5786.262} C_VEL
LIN {X 0,Y 650.663,Z 707.31,A -85,B 0,C 180,E1 5790.825,E2 5790.825} C_VEL
LIN {X 0,Y 650.695,Z 707.31,A -85,B 0,C 180,E1 5795.61,E2 5795.61} C_VEL
LIN {X 0,Y 650.803,Z 707.31,A -85,B 0,C 180,E1 5800.694,E2 5800.694} C_VEL
LIN {X 0,Y 650.729,Z 707.31,A -85,B 0,C 180,E1 5806.216,E2 5806.216} C_VEL
LIN {X 0,Y 650.812,Z 707.31,A -85,B 0,C 180,E1 5811.047,E2 5811.047} C_VEL
LIN {X 0,Y 650.868,Z 707.31,A -85,B 0,C 180,E1 5813.027,E2 5813.027} C_VEL
LIN {X 0,Y 667.897,Z 746.508,A -85,B 0,C 180,E1 5814.616,E2 5814.616} C_VEL
LIN {X 0,Y 666.192,Z 792.051,A -85,B 0,C 180,E1 5815.66,E2 5815.66} C_VEL
LIN {X 0,Y 663.682,Z 838.286,A -85,B 0,C 180,E1 5817.342,E2 5817.342} C_VEL
LIN {X 0,Y 660.903,Z 881.888,A -85,B 0,C 180,E1 5819.596,E2 5819.596} C_VEL
LIN {X 0,Y 658.109,Z 921.328,A -85,B 0,C 180,E1 5822.315,E2 5822.315} C_VEL
LIN {X 0,Y 655.811,Z 956.032,A -85,B 0,C 180,E1 5825.423,E2 5825.423} C_VEL
LIN {X 0,Y 653.956,Z 985.3,A -85,B 0,C 180,E1 5828.773,E2 5828.773} C_VEL
LIN {X 0,Y 652.77,Z 1010.009,A -85,B 0,C 180,E1 5832.435,E2 5832.435} C_VEL
LIN {X 0,Y 652.047,Z 1029.125,A -85,B 0,C 180,E1 5836.219,E2 5836.219} C_VEL
LIN {X 0,Y 651.693,Z 1042.22,A -85,B 0,C 180,E1 5839.957,E2 5839.957} C_VEL
LIN {X 0,Y 651.587,Z 1049.731,A -85,B 0,C 180,E1 5843.323,E2 5843.323} C_VEL
LIN {X 0,Y 651.435,Z 1053.351,A -85,B 0,C 180,E1 5847.334,E2 5847.334} C_VEL
LIN {X 0,Y 651.543,Z 1051.449,A -85,B 0,C 180,E1 5851.333,E2 5851.333} C_VEL
LIN {X 0,Y 651.583,Z 1043.979,A -85,B 0,C 180,E1 5855.338,E2 5855.338} C_VEL
LIN {X 0,Y 651.812,Z 1032.274,A -85,B 0,C 180,E1 5858.902,E2 5858.902} C_VEL
LIN {X 0,Y 652.443,Z 1014.463,A -85,B 0,C 180,E1 5862.698,E2 5862.698} C_VEL
LIN {X 0,Y 653.668,Z 990.19,A -85,B 0,C 180,E1 5866.499,E2 5866.499} C_VEL
LIN {X 0,Y 655.519,Z 959.781,A -85,B 0,C 180,E1 5870.114,E2 5870.114} C_VEL
LIN {X 0,Y 658.034,Z 923.713,A -85,B 0,C 180,E1 5873.407,E2 5873.407} C_VEL
LIN {X 0,Y 660.896,Z 882.964,A -85,B 0,C 180,E1 5876.248,E2 5876.248} C_VEL
LIN {X 0,Y 663.785,Z 838.846,A -85,B 0,C 180,E1 5878.537,E2 5878.537} C_VEL
LIN {X 0,Y 666.028,Z 794.964,A -85,B 0,C 180,E1 5880.159,E2 5880.159} C_VEL
LIN {X 0,Y 667.779,Z 752.79,A -85,B 0,C 180,E1 5881.176,E2 5881.176} C_VEL
LIN {X 0,Y 667.123,Z 742.729,A -85,B 0,C 180,E1 5881.412,E2 5881.412} C_VEL
LIN {X 0,Y 650.729,Z 707.31,A -85,B 0,C 180,E1 5882.929,E2 5882.929} C_VEL
LIN {X 0,Y 650.73,Z 707.31,A -85,B 0,C 180,E1 5887.645,E2 5887.645} C_VEL
LIN {X 0,Y 650.686,Z 707.31,A -85,B 0,C 180,E1 5892.485,E2 5892.485} C_VEL
LIN {X 0,Y 650.805,Z 707.31,A -85,B 0,C 180,E1 5898.17,E2 5898.17} C_VEL
LIN {X 0,Y 650.746,Z 707.31,A -85,B 0,C 180,E1 5902.735,E2 5902.735} C_VEL
LIN {X 0,Y 650.826,Z 707.31,A -85,B 0,C 180,E1 5907.617,E2 5907.617} C_VEL
LIN {X 0,Y 650.858,Z 707.31,A -85,B 0,C 180,E1 5912.245,E2 5912.245} C_VEL
LIN {X 0,Y 650.802,Z 707.31,A -85,B 0,C 180,E1 5918.124,E2 5918.124} C_VEL
LIN {X 0,Y 650.862,Z 707.31,A -85,B 0,C 180,E1 5923.774,E2 5923.774} C_VEL
LIN {X 0,Y 651.266,Z 707.31,A -85,B 0,C 180,E1 5927.91,E2 5927.91} C_VEL
LIN {X 0,Y 651.214,Z 707.31,A -85,B 0,C 180,E1 5933.316,E2 5933.316} C_VEL
LIN {X 0,Y 650.887,Z 707.31,A -85,B 0,C 180,E1 5937.329,E2 5937.329} C_VEL
LIN {X 0,Y 651.435,Z 707.31,A -85,B 0,C 180,E1 5941.331,E2 5941.331} C_VEL
LIN {X 0,Y 651.332,Z 707.31,A -85,B 0,C 180,E1 5948.022,E2 5948.022} C_VEL
LIN {X 0,Y 651.024,Z 707.31,A -85,B 0,C 180,E1 5953.458,E2 5953.458} C_VEL
LIN {X 0,Y 650.85,Z 707.31,A -85,B 0,C 180,E1 5959.021,E2 5959.021} C_VEL
LIN {X 0,Y 650.784,Z 707.31,A -85,B 0,C 180,E1 5964.778,E2 5964.778} C_VEL
LIN {X 0,Y 650.899,Z 707.31,A -85,B 0,C 180,E1 5970.523,E2 5970.523} C_VEL
LIN {X 0,Y 650.798,Z 707.31,A -85,B 0,C 180,E1 5973.311,E2 5973.311} C_VEL
LIN {X 0,Y 646.831,Z 707.31,A -85,B 0,C 180,E1 5974.808,E2 5974.808} C_VEL
LIN {X 0,Y 642.835,Z 707.31,A -85,B 0,C 180,E1 5976.323,E2 5976.323} C_VEL
LIN {X 0,Y 642.8,Z 707.31,A -85,B 0,C 180,E1 5981.304,E2 5981.304} C_VEL
LIN {X 0,Y 642.766,Z 707.31,A -85,B 0,C 180,E1 5986.954,E2 5986.954} C_VEL
LIN {X 0,Y 642.786,Z 707.31,A -85,B 0,C 180,E1 5992.195,E2 5992.195} C_VEL
LIN {X 0,Y 642.854,Z 708.099,A -85,B 0,C 180,E1 5994.209,E2 5994.209} C_VEL
LIN {X 0,Y 661.745,Z 749.32,A -85,B 0,C 180,E1 5995.901,E2 5995.901} C_VEL
LIN {X 0,Y 660.37,Z 798.387,A -85,B 0,C 180,E1 5996.722,E2 5996.722} C_VEL
LIN {X 0,Y 658.348,Z 843.02,A -85,B 0,C 180,E1 5998.033,E2 5998.033} C_VEL
LIN {X 0,Y 655.708,Z 885.396,A -85,B 0,C 180,E1 5999.841,E2 5999.841} C_VEL
LIN {X 0,Y 652.674,Z 927.893,A -85,B 0,C 180,E1 6002.33,E2 6002.33} C_VEL
LIN {X 0,Y 649.639,Z 967.309,A -85,B 0,C 180,E1 6005.394,E2 6005.394} C_VEL
LIN {X 0,Y 647.166,Z 1001.737,A -85,B 0,C 180,E1 6008.898,E2 6008.898} C_VEL
LIN {X 0,Y 645.362,Z 1030.655,A -85,B 0,C 180,E1 6012.755,E2 6012.755} C_VEL
LIN {X 0,Y 644.404,Z 1053.258,A -85,B 0,C 180,E1 6016.806,E2 6016.806} C_VEL
LIN {X 0,Y 643.917,Z 1069.573,A -85,B 0,C 180,E1 6020.982,E2 6020.982} C_VEL
LIN {X 0,Y 643.675,Z 1078.458,A -85,B 0,C 180,E1 6024.596,E2 6024.596} C_VEL
LIN {X 0,Y 643.603,Z 1083.167,A -85,B 0,C 180,E1 6028.65,E2 6028.65} C_VEL
LIN {X 0,Y 643.75,Z 1082.216,A -85,B 0,C 180,E1 6032.698,E2 6032.698} C_VEL
LIN {X 0,Y 643.676,Z 1075.636,A -85,B 0,C 180,E1 6036.76,E2 6036.76} C_VEL
LIN {X 0,Y 643.921,Z 1064.514,A -85,B 0,C 180,E1 6040.508,E2 6040.508} C_VEL
LIN {X 0,Y 644.678,Z 1046.036,A -85,B 0,C 180,E1 6044.636,E2 6044.636} C_VEL
LIN {X 0,Y 646.045,Z 1020.442,A -85,B 0,C 180,E1 6048.736,E2 6048.736} C_VEL
LIN {X 0,Y 648.006,Z 989.87,A -85,B 0,C 180,E1 6052.42,E2 6052.42} C_VEL
LIN {X 0,Y 650.718,Z 953.251,A -85,B 0,C 180,E1 6055.797,E2 6055.797} C_VEL
LIN {X 0,Y 653.763,Z 913.212,A -85,B 0,C 180,E1 6058.616,E2 6058.616} C_VEL
LIN {X 0,Y 656.772,Z 869.719,A -85,B 0,C 180,E1 6060.902,E2 6060.902} C_VEL
LIN {X 0,Y 659.428,Z 822.389,A -85,B 0,C 180,E1 6062.649,E2 6062.649} C_VEL
LIN {X 0,Y 661.241,Z 773.535,A -85,B 0,C 180,E1 6063.77,E2 6063.77} C_VEL
LIN {X 0,Y 661.212,Z 746.179,A -85,B 0,C 180,E1 6064.17,E2 6064.17} C_VEL
LIN {X 0,Y 642.884,Z 707.31,A -85,B 0,C 180,E1 6065.825,E2 6065.825} C_VEL
LIN {X 0,Y 642.853,Z 707.31,A -85,B 0,C 180,E1 6071.302,E2 6071.302} C_VEL
LIN {X 0,Y 642.762,Z 707.31,A -85,B 0,C 180,E1 6076.958,E2 6076.958} C_VEL
LIN {X 0,Y 642.817,Z 707.31,A -85,B 0,C 180,E1 6082.202,E2 6082.202} C_VEL
LIN {X 0,Y 642.925,Z 707.31,A -85,B 0,C 180,E1 6088.051,E2 6088.051} C_VEL
LIN {X 0,Y 642.978,Z 707.31,A -85,B 0,C 180,E1 6093.584,E2 6093.584} C_VEL
LIN {X 0,Y 642.932,Z 707.31,A -85,B 0,C 180,E1 6099.298,E2 6099.298} C_VEL
LIN {X 0,Y 643.074,Z 707.31,A -85,B 0,C 180,E1 6105.05,E2 6105.05} C_VEL
LIN {X 0,Y 643.355,Z 707.31,A -85,B 0,C 180,E1 6110.512,E2 6110.512} C_VEL
LIN {X 0,Y 643.126,Z 707.31,A -85,B 0,C 180,E1 6114.594,E2 6114.594} C_VEL
LIN {X 0,Y 643.269,Z 707.31,A -85,B 0,C 180,E1 6120.002,E2 6120.002} C_VEL
LIN {X 0,Y 643.266,Z 707.31,A -85,B 0,C 180,E1 6125.409,E2 6125.409} C_VEL
LIN {X 0,Y 643.209,Z 707.31,A -85,B 0,C 180,E1 6130.866,E2 6130.866} C_VEL
LIN {X 0,Y 642.931,Z 707.31,A -85,B 0,C 180,E1 6136.432,E2 6136.432} C_VEL
LIN {X 0,Y 643.074,Z 707.31,A -85,B 0,C 180,E1 6142.153,E2 6142.153} C_VEL
LIN {X 0,Y 642.835,Z 707.31,A -85,B 0,C 180,E1 6146.611,E2 6146.611} C_VEL
LIN {X 0,Y 642.706,Z 707.31,A -85,B 0,C 180,E1 6151.917,E2 6151.917} C_VEL
LIN {X 0,Y 642.796,Z 707.31,A -85,B 0,C 180,E1 6157.806,E2 6157.806} C_VEL
LIN {X 0,Y 642.849,Z 707.31,A -85,B 0,C 180,E1 6163.13,E2 6163.13} C_VEL
LIN {X 0,Y 642.845,Z 707.31,A -85,B 0,C 180,E1 6168.971,E2 6168.971} C_VEL
LIN {X 0,Y 642.945,Z 707.31,A -85,B 0,C 180,E1 6172.515,E2 6172.515} C_VEL
LIN {X 0,Y 661.228,Z 747.823,A -85,B 0,C 180,E1 6174.257,E2 6174.257} C_VEL
LIN {X 0,Y 659.482,Z 792.387,A -85,B 0,C 180,E1 6175.296,E2 6175.296} C_VEL
LIN {X 0,Y 656.76,Z 838.835,A -85,B 0,C 180,E1 6177.009,E2 6177.009} C_VEL
LIN {X 0,Y 653.704,Z 883.219,A -85,B 0,C 180,E1 6179.337,E2 6179.337} C_VEL
LIN {X 0,Y 650.556,Z 924.73,A -85,B 0,C 180,E1 6182.276,E2 6182.276} C_VEL
LIN {X 0,Y 648.003,Z 959.949,A -85,B 0,C 180,E1 6185.544,E2 6185.544} C_VEL
LIN {X 0,Y 646.031,Z 990.456,A -85,B 0,C 180,E1 6189.22,E2 6189.22} C_VEL
LIN {X 0,Y 644.652,Z 1015.761,A -85,B 0,C 180,E1 6193.265,E2 6193.265} C_VEL
LIN {X 0,Y 644.018,Z 1034.168,A -85,B 0,C 180,E1 6197.36,E2 6197.36} C_VEL
LIN {X 0,Y 643.691,Z 1045.311,A -85,B 0,C 180,E1 6201.055,E2 6201.055} C_VEL
LIN {X 0,Y 643.64,Z 1051.527,A -85,B 0,C 180,E1 6204.597,E2 6204.597} C_VEL
LIN {X 0,Y 643.574,Z 1053.333,A -85,B 0,C 180,E1 6208.651,E2 6208.651} C_VEL
LIN {X 0,Y 643.676,Z 1049.633,A -85,B 0,C 180,E1 6212.699,E2 6212.699} C_VEL
LIN {X 0,Y 643.875,Z 1040.219,A -85,B 0,C 180,E1 6216.759,E2 6216.759} C_VEL
LIN {X 0,Y 644.332,Z 1024.62,A -85,B 0,C 180,E1 6220.846,E2 6220.846} C_VEL
LIN {X 0,Y 645.251,Z 1003.173,A -85,B 0,C 180,E1 6224.798,E2 6224.798} C_VEL
LIN {X 0,Y 646.817,Z 977.145,A -85,B 0,C 180,E1 6228.406,E2 6228.406} C_VEL
LIN {X 0,Y 649.039,Z 945.919,A -85,B 0,C 180,E1 6231.763,E2 6231.763} C_VEL
LIN {X 0,Y 651.762,Z 908.944,A -85,B 0,C 180,E1 6234.848,E2 6234.848} C_VEL
LIN {X 0,Y 654.878,Z 867.733,A -85,B 0,C 180,E1 6237.465,E2 6237.465} C_VEL
LIN {X 0,Y 657.797,Z 822.181,A -85,B 0,C 180,E1 6239.592,E2 6239.592} C_VEL
LIN {X 0,Y 660.156,Z 776.467,A -85,B 0,C 180,E1 6241.054,E2 6241.054} C_VEL
LIN {X 0,Y 660.799,Z 746.084,A -85,B 0,C 180,E1 6241.713,E2 6241.713} C_VEL
LIN {X 0,Y 642.796,Z 707.31,A -85,B 0,C 180,E1 6243.471,E2 6243.471} C_VEL
LIN {X 0,Y 642.845,Z 707.31,A -85,B 0,C 180,E1 6249.531,E2 6249.531} C_VEL
LIN {X 0,Y 642.843,Z 707.31,A -85,B 0,C 180,E1 6255.009,E2 6255.009} C_VEL
LIN {X 0,Y 642.872,Z 707.31,A -85,B 0,C 180,E1 6260.47,E2 6260.47} C_VEL
LIN {X 0,Y 642.87,Z 707.31,A -85,B 0,C 180,E1 6265.593,E2 6265.593} C_VEL
LIN {X 0,Y 642.953,Z 707.31,A -85,B 0,C 180,E1 6270.701,E2 6270.701} C_VEL
LIN {X 0,Y 642.89,Z 707.31,A -85,B 0,C 180,E1 6274.892,E2 6274.892} C_VEL
LIN {X 0,Y 642.921,Z 707.31,A -85,B 0,C 180,E1 6280.73,E2 6280.73} C_VEL
LIN {X 0,Y 643.304,Z 707.31,A -85,B 0,C 180,E1 6286.373,E2 6286.373} C_VEL
LIN {X 0,Y 643.332,Z 707.31,A -85,B 0,C 180,E1 6291.873,E2 6291.873} C_VEL
LIN {X 0,Y 643.289,Z 707.31,A -85,B 0,C 180,E1 6295.945,E2 6295.945} C_VEL
LIN {X 0,Y 643.522,Z 707.31,A -85,B 0,C 180,E1 6301.347,E2 6301.347} C_VEL
LIN {X 0,Y 643.415,Z 707.31,A -85,B 0,C 180,E1 6308.121,E2 6308.121} C_VEL
LIN {X 0,Y 643.101,Z 707.31,A -85,B 0,C 180,E1 6313.627,E2 6313.627} C_VEL
LIN {X 0,Y 642.919,Z 707.31,A -85,B 0,C 180,E1 6319.467,E2 6319.467} C_VEL
LIN {X 0,Y 642.869,Z 707.31,A -85,B 0,C 180,E1 6325.104,E2 6325.104} C_VEL
LIN {X 0,Y 642.924,Z 707.31,A -85,B 0,C 180,E1 6329.665,E2 6329.665} C_VEL
LIN {X 0,Y 642.888,Z 707.31,A -85,B 0,C 180,E1 6334.449,E2 6334.449} C_VEL
LIN {X 0,Y 642.835,Z 707.31,A -85,B 0,C 180,E1 6336.323,E2 6336.323} C_VEL
LIN {X 0,Y 638.81,Z 707.31,A -85,B 0,C 180,E1 6337.85,E2 6337.85} C_VEL
LIN {X 0,Y 634.818,Z 707.31,A -85,B 0,C 180,E1 6339.396,E2 6339.396} C_VEL
LIN {X 0,Y 634.804,Z 707.31,A -85,B 0,C 180,E1 6344.261,E2 6344.261} C_VEL
LIN {X 0,Y 634.855,Z 707.31,A -85,B 0,C 180,E1 6349.872,E2 6349.872} C_VEL
LIN {X 0,Y 634.864,Z 707.31,A -85,B 0,C 180,E1 6353.659,E2 6353.659} C_VEL
LIN {X 0,Y 655.167,Z 751.776,A -85,B 0,C 180,E1 6355.546,E2 6355.546} C_VEL
LIN {X 0,Y 653.617,Z 801.087,A -85,B 0,C 180,E1 6356.406,E2 6356.406} C_VEL
LIN {X 0,Y 651.345,Z 846.077,A -85,B 0,C 180,E1 6357.78,E2 6357.78} C_VEL
LIN {X 0,Y 648.452,Z 888.804,A -85,B 0,C 180,E1 6359.665,E2 6359.665} C_VEL
LIN {X 0,Y 645.399,Z 929.156,A -85,B 0,C 180,E1 6362.086,E2 6362.086} C_VEL
LIN {X 0,Y 642.266,Z 966.725,A -85,B 0,C 180,E1 6365.036,E2 6365.036} C_VEL
LIN {X 0,Y 639.582,Z 1001.739,A -85,B 0,C 180,E1 6368.636,E2 6368.636} C_VEL
LIN {X 0,Y 637.616,Z 1030.657,A -85,B 0,C 180,E1 6372.539,E2 6372.539} C_VEL
LIN {X 0,Y 636.559,Z 1052.974,A -85,B 0,C 180,E1 6376.576,E2 6376.576} C_VEL
LIN {X 0,Y 636.037,Z 1069.303,A -85,B 0,C 180,E1 6380.788,E2 6380.788} C_VEL
LIN {X 0,Y 635.781,Z 1078.458,A -85,B 0,C 180,E1 6384.528,E2 6384.528} C_VEL
LIN {X 0,Y 635.709,Z 1083.166,A -85,B 0,C 180,E1 6388.633,E2 6388.633} C_VEL
LIN {X 0,Y 635.877,Z 1082.216,A -85,B 0,C 180,E1 6392.731,E2 6392.731} C_VEL
LIN {X 0,Y 635.801,Z 1075.636,A -85,B 0,C 180,E1 6396.844,E2 6396.844} C_VEL
LIN {X 0,Y 636.153,Z 1063.176,A -85,B 0,C 180,E1 6400.985,E2 6400.985} C_VEL
LIN {X 0,Y 636.889,Z 1046.037,A -85,B 0,C 180,E1 6404.819,E2 6404.819} C_VEL
LIN {X 0,Y 638.344,Z 1020.922,A -85,B 0,C 180,E1 6408.901,E2 6408.901} C_VEL
LIN {X 0,Y 640.449,Z 990.133,A -85,B 0,C 180,E1 6412.669,E2 6412.669} C_VEL
LIN {X 0,Y 643.418,Z 953.253,A -85,B 0,C 180,E1 6416.112,E2 6416.112} C_VEL
LIN {X 0,Y 646.687,Z 912.983,A -85,B 0,C 180,E1 6418.973,E2 6418.973} C_VEL
LIN {X 0,Y 649.911,Z 868.858,A -85,B 0,C 180,E1 6421.299,E2 6421.299} C_VEL
LIN {X 0,Y 652.727,Z 821.887,A -85,B 0,C 180,E1 6423.036,E2 6423.036} C_VEL
LIN {X 0,Y 654.669,Z 773.313,A -85,B 0,C 180,E1 6424.155,E2 6424.155} C_VEL
LIN {X 0,Y 654.429,Z 748.437,A -85,B 0,C 180,E1 6424.541,E2 6424.541} C_VEL
LIN {X 0,Y 634.942,Z 707.31,A -85,B 0,C 180,E1 6426.341,E2 6426.341} C_VEL
LIN {X 0,Y 634.864,Z 707.31,A -85,B 0,C 180,E1 6432.276,E2 6432.276} C_VEL
LIN {X 0,Y 634.808,Z 707.31,A -85,B 0,C 180,E1 6438.06,E2 6438.06} C_VEL
LIN {X 0,Y 634.937,Z 707.31,A -85,B 0,C 180,E1 6443.372,E2 6443.372} C_VEL
LIN {X 0,Y 634.979,Z 707.31,A -85,B 0,C 180,E1 6449.22,E2 6449.22} C_VEL
LIN {X 0,Y 634.976,Z 707.31,A -85,B 0,C 180,E1 6454.562,E2 6454.562} C_VEL
LIN {X 0,Y 635.015,Z 707.31,A -85,B 0,C 180,E1 6460.485,E2 6460.485} C_VEL
LIN {X 0,Y 635.175,Z 707.31,A -85,B 0,C 180,E1 6466.2,E2 6466.2} C_VEL
LIN {X 0,Y 635.509,Z 707.31,A -85,B 0,C 180,E1 6471.777,E2 6471.777} C_VEL
LIN {X 0,Y 635.593,Z 707.31,A -85,B 0,C 180,E1 6478.636,E2 6478.636} C_VEL
LIN {X 0,Y 635.336,Z 707.31,A -85,B 0,C 180,E1 6485.477,E2 6485.477} C_VEL
LIN {X 0,Y 635.29,Z 707.31,A -85,B 0,C 180,E1 6491.004,E2 6491.004} C_VEL
LIN {X 0,Y 635.002,Z 707.31,A -85,B 0,C 180,E1 6496.643,E2 6496.643} C_VEL
LIN {X 0,Y 635.15,Z 707.31,A -85,B 0,C 180,E1 6502.444,E2 6502.444} C_VEL
LIN {X 0,Y 634.843,Z 707.31,A -85,B 0,C 180,E1 6507.97,E2 6507.97} C_VEL
LIN {X 0,Y 634.813,Z 707.31,A -85,B 0,C 180,E1 6513.333,E2 6513.333} C_VEL
LIN {X 0,Y 634.893,Z 707.31,A -85,B 0,C 180,E1 6518.361,E2 6518.361} C_VEL
LIN {X 0,Y 634.86,Z 707.31,A -85,B 0,C 180,E1 6524.268,E2 6524.268} C_VEL
LIN {X 0,Y 634.923,Z 707.31,A -85,B 0,C 180,E1 6529.879,E2 6529.879} C_VEL
LIN {X 0,Y 635.03,Z 707.718,A -85,B 0,C 180,E1 6532.028,E2 6532.028} C_VEL
LIN {X 0,Y 654.583,Z 751.842,A -85,B 0,C 180,E1 6533.946,E2 6533.946} C_VEL
LIN {X 0,Y 652.68,Z 795.137,A -85,B 0,C 180,E1 6535.003,E2 6535.003} C_VEL
LIN {X 0,Y 649.861,Z 839.813,A -85,B 0,C 180,E1 6536.683,E2 6536.683} C_VEL
LIN {X 0,Y 646.514,Z 884.224,A -85,B 0,C 180,E1 6539.057,E2 6539.057} C_VEL
LIN {X 0,Y 643.207,Z 924.986,A -85,B 0,C 180,E1 6541.984,E2 6541.984} C_VEL
LIN {X 0,Y 640.422,Z 960.833,A -85,B 0,C 180,E1 6545.364,E2 6545.364} C_VEL
LIN {X 0,Y 638.255,Z 991.505,A -85,B 0,C 180,E1 6549.137,E2 6549.137} C_VEL
LIN {X 0,Y 636.864,Z 1015.708,A -85,B 0,C 180,E1 6553.071,E2 6553.071} C_VEL
LIN {X 0,Y 636.141,Z 1034.337,A -85,B 0,C 180,E1 6557.271,E2 6557.271} C_VEL
LIN {X 0,Y 635.777,Z 1046.122,A -85,B 0,C 180,E1 6561.325,E2 6561.325} C_VEL
LIN {X 0,Y 635.735,Z 1051.496,A -85,B 0,C 180,E1 6564.529,E2 6564.529} C_VEL
LIN {X 0,Y 635.696,Z 1053.339,A -85,B 0,C 180,E1 6568.635,E2 6568.635} C_VEL
LIN {X 0,Y 635.784,Z 1049.678,A -85,B 0,C 180,E1 6572.733,E2 6572.733} C_VEL
LIN {X 0,Y 636,Z 1040.291,A -85,B 0,C 180,E1 6576.843,E2 6576.843} C_VEL
LIN {X 0,Y 636.475,Z 1024.738,A -85,B 0,C 180,E1 6580.981,E2 6580.981} C_VEL
LIN {X 0,Y 637.429,Z 1004.412,A -85,B 0,C 180,E1 6584.808,E2 6584.808} C_VEL
LIN {X 0,Y 639.068,Z 978.778,A -85,B 0,C 180,E1 6588.462,E2 6588.462} C_VEL
LIN {X 0,Y 641.562,Z 946.273,A -85,B 0,C 180,E1 6592.023,E2 6592.023} C_VEL
LIN {X 0,Y 644.512,Z 909.323,A -85,B 0,C 180,E1 6595.147,E2 6595.147} C_VEL
LIN {X 0,Y 647.88,Z 867.547,A -85,B 0,C 180,E1 6597.827,E2 6597.827} C_VEL
LIN {X 0,Y 651.007,Z 823.009,A -85,B 0,C 180,E1 6599.936,E2 6599.936} C_VEL
LIN {X 0,Y 653.598,Z 776.008,A -85,B 0,C 180,E1 6601.448,E2 6601.448} C_VEL
LIN {X 0,Y 654.246,Z 748.905,A -85,B 0,C 180,E1 6602.044,E2 6602.044} C_VEL
LIN {X 0,Y 634.883,Z 707.31,A -85,B 0,C 180,E1 6603.942,E2 6603.942} C_VEL
LIN {X 0,Y 634.902,Z 707.31,A -85,B 0,C 180,E1 6608.359,E2 6608.359} C_VEL
LIN {X 0,Y 634.823,Z 707.31,A -85,B 0,C 180,E1 6614.261,E2 6614.261} C_VEL
LIN {X 0,Y 634.931,Z 707.31,A -85,B 0,C 180,E1 6619.876,E2 6619.876} C_VEL
LIN {X 0,Y 634.898,Z 707.31,A -85,B 0,C 180,E1 6625.049,E2 6625.049} C_VEL
LIN {X 0,Y 634.976,Z 707.31,A -85,B 0,C 180,E1 6629.92,E2 6629.92} C_VEL
LIN {X 0,Y 634.985,Z 707.31,A -85,B 0,C 180,E1 6635.078,E2 6635.078} C_VEL
LIN {X 0,Y 635.021,Z 707.31,A -85,B 0,C 180,E1 6640.48,E2 6640.48} C_VEL
LIN {X 0,Y 635.362,Z 707.31,A -85,B 0,C 180,E1 6646.199,E2 6646.199} C_VEL
LIN {X 0,Y 635.434,Z 707.31,A -85,B 0,C 180,E1 6651.844,E2 6651.844} C_VEL
LIN {X 0,Y 635.405,Z 707.31,A -85,B 0,C 180,E1 6655.895,E2 6655.895} C_VEL
LIN {X 0,Y 635.608,Z 707.31,A -85,B 0,C 180,E1 6661.364,E2 6661.364} C_VEL
LIN {X 0,Y 635.518,Z 707.31,A -85,B 0,C 180,E1 6668.223,E2 6668.223} C_VEL
LIN {X 0,Y 635.186,Z 707.31,A -85,B 0,C 180,E1 6673.8,E2 6673.8} C_VEL
LIN {X 0,Y 635.019,Z 707.31,A -85,B 0,C 180,E1 6679.515,E2 6679.515} C_VEL
LIN {X 0,Y 634.986,Z 707.31,A -85,B 0,C 180,E1 6685.437,E2 6685.437} C_VEL
LIN {X 0,Y 634.984,Z 707.31,A -85,B 0,C 180,E1 6690.778,E2 6690.778} C_VEL
LIN {X 0,Y 634.947,Z 707.31,A -85,B 0,C 180,E1 6696.628,E2 6696.628} C_VEL
LIN {X 0,Y 634.818,Z 707.31,A -85,B 0,C 180,E1 6699.396,E2 6699.396} C_VEL
LIN {X 0,Y 630.816,Z 707.31,A -85,B 0,C 180,E1 6700.942,E2 6700.942} C_VEL
LIN {X 0,Y 626.872,Z 707.31,A -85,B 0,C 180,E1 6702.507,E2 6702.507} C_VEL
LIN {X 0,Y 626.871,Z 707.31,A -85,B 0,C 180,E1 6707.399,E2 6707.399} C_VEL
LIN {X 0,Y 626.973,Z 707.31,A -85,B 0,C 180,E1 6713.133,E2 6713.133} C_VEL
LIN {X 0,Y 648.629,Z 754.388,A -85,B 0,C 180,E1 6715.186,E2 6715.186} C_VEL
LIN {X 0,Y 646.83,Z 805.103,A -85,B 0,C 180,E1 6716.115,E2 6716.115} C_VEL
LIN {X 0,Y 643.958,Z 854.288,A -85,B 0,C 180,E1 6717.715,E2 6717.715} C_VEL
LIN {X 0,Y 640.579,Z 899.623,A -85,B 0,C 180,E1 6719.889,E2 6719.889} C_VEL
LIN {X 0,Y 637.184,Z 940.532,A -85,B 0,C 180,E1 6722.561,E2 6722.561} C_VEL
LIN {X 0,Y 633.871,Z 979.133,A -85,B 0,C 180,E1 6725.907,E2 6725.907} C_VEL
LIN {X 0,Y 631.252,Z 1011.107,A -85,B 0,C 180,E1 6729.524,E2 6729.524} C_VEL
LIN {X 0,Y 629.498,Z 1038.167,A -85,B 0,C 180,E1 6733.554,E2 6733.554} C_VEL
LIN {X 0,Y 628.463,Z 1059.13,A -85,B 0,C 180,E1 6737.819,E2 6737.819} C_VEL
LIN {X 0,Y 628.072,Z 1072.156,A -85,B 0,C 180,E1 6741.676,E2 6741.676} C_VEL
LIN {X 0,Y 627.922,Z 1079.664,A -85,B 0,C 180,E1 6745.154,E2 6745.154} C_VEL
LIN {X 0,Y 627.808,Z 1083.166,A -85,B 0,C 180,E1 6748.616,E2 6748.616} C_VEL
LIN {X 0,Y 627.973,Z 1082.215,A -85,B 0,C 180,E1 6752.766,E2 6752.766} C_VEL
LIN {X 0,Y 627.908,Z 1075.636,A -85,B 0,C 180,E1 6756.93,E2 6756.93} C_VEL
LIN {X 0,Y 628.313,Z 1063.175,A -85,B 0,C 180,E1 6761.124,E2 6761.124} C_VEL
LIN {X 0,Y 629.088,Z 1046.038,A -85,B 0,C 180,E1 6765.007,E2 6765.007} C_VEL
LIN {X 0,Y 630.652,Z 1021.128,A -85,B 0,C 180,E1 6769.11,E2 6769.11} C_VEL
LIN {X 0,Y 632.932,Z 990.134,A -85,B 0,C 180,E1 6772.954,E2 6772.954} C_VEL
LIN {X 0,Y 636.081,Z 953.486,A -85,B 0,C 180,E1 6776.417,E2 6776.417} C_VEL
LIN {X 0,Y 639.543,Z 913.415,A -85,B 0,C 180,E1 6779.292,E2 6779.292} C_VEL
LIN {X 0,Y 643.022,Z 868.823,A -85,B 0,C 180,E1 6781.664,E2 6781.664} C_VEL
LIN {X 0,Y 646.073,Z 821.567,A -85,B 0,C 180,E1 6783.425,E2 6783.425} C_VEL
LIN {X 0,Y 648.121,Z 773.408,A -85,B 0,C 180,E1 6784.543,E2 6784.543} C_VEL
LIN {X 0,Y 647.861,Z 750.903,A -85,B 0,C 180,E1 6784.907,E2 6784.907} C_VEL
LIN {X 0,Y 627.027,Z 707.31,A -85,B 0,C 180,E1 6786.936,E2 6786.936} C_VEL
LIN {X 0,Y 626.924,Z 707.31,A -85,B 0,C 180,E1 6792.594,E2 6792.594} C_VEL
LIN {X 0,Y 626.869,Z 707.31,A -85,B 0,C 180,E1 6797.404,E2 6797.404} C_VEL
LIN {X 0,Y 627.006,Z 707.31,A -85,B 0,C 180,E1 6802.898,E2 6802.898} C_VEL
LIN {X 0,Y 627.059,Z 707.31,A -85,B 0,C 180,E1 6807.885,E2 6807.885} C_VEL
LIN {X 0,Y 627.085,Z 707.31,A -85,B 0,C 180,E1 6813.396,E2 6813.396} C_VEL
LIN {X 0,Y 627.056,Z 707.31,A -85,B 0,C 180,E1 6818.749,E2 6818.749} C_VEL
LIN {X 0,Y 627.196,Z 707.31,A -85,B 0,C 180,E1 6824.59,E2 6824.59} C_VEL
LIN {X 0,Y 627.521,Z 707.31,A -85,B 0,C 180,E1 6830.27,E2 6830.27} C_VEL
LIN {X 0,Y 627.337,Z 707.31,A -85,B 0,C 180,E1 6834.458,E2 6834.458} C_VEL
LIN {X 0,Y 627.463,Z 707.31,A -85,B 0,C 180,E1 6840.003,E2 6840.003} C_VEL
LIN {X 0,Y 627.406,Z 707.31,A -85,B 0,C 180,E1 6845.547,E2 6845.547} C_VEL
LIN {X 0,Y 627.375,Z 707.31,A -85,B 0,C 180,E1 6851.144,E2 6851.144} C_VEL
LIN {X 0,Y 627.083,Z 707.31,A -85,B 0,C 180,E1 6856.86,E2 6856.86} C_VEL
LIN {X 0,Y 627.246,Z 707.31,A -85,B 0,C 180,E1 6861.25,E2 6861.25} C_VEL
LIN {X 0,Y 626.974,Z 707.31,A -85,B 0,C 180,E1 6866.584,E2 6866.584} C_VEL
LIN {X 0,Y 626.884,Z 707.31,A -85,B 0,C 180,E1 6872.214,E2 6872.214} C_VEL
LIN {X 0,Y 626.947,Z 707.31,A -85,B 0,C 180,E1 6877.179,E2 6877.179} C_VEL
LIN {X 0,Y 626.957,Z 707.31,A -85,B 0,C 180,E1 6882.595,E2 6882.595} C_VEL
LIN {X 0,Y 626.911,Z 707.31,A -85,B 0,C 180,E1 6888.537,E2 6888.537} C_VEL
LIN {X 0,Y 627.102,Z 707.665,A -85,B 0,C 180,E1 6891.493,E2 6891.493} C_VEL
LIN {X 0,Y 647.998,Z 753.363,A -85,B 0,C 180,E1 6893.58,E2 6893.58} C_VEL
LIN {X 0,Y 645.988,Z 795.863,A -85,B 0,C 180,E1 6894.636,E2 6894.636} C_VEL
LIN {X 0,Y 642.959,Z 841.146,A -85,B 0,C 180,E1 6896.368,E2 6896.368} C_VEL
LIN {X 0,Y 639.49,Z 884.032,A -85,B 0,C 180,E1 6898.687,E2 6898.687} C_VEL
LIN {X 0,Y 635.968,Z 924.625,A -85,B 0,C 180,E1 6901.633,E2 6901.633} C_VEL
LIN {X 0,Y 632.904,Z 960.975,A -85,B 0,C 180,E1 6905.097,E2 6905.097} C_VEL
LIN {X 0,Y 630.641,Z 991.32,A -85,B 0,C 180,E1 6908.873,E2 6908.873} C_VEL
LIN {X 0,Y 629.101,Z 1015.708,A -85,B 0,C 180,E1 6912.883,E2 6912.883} C_VEL
LIN {X 0,Y 628.277,Z 1034.235,A -85,B 0,C 180,E1 6917.109,E2 6917.109} C_VEL
LIN {X 0,Y 627.915,Z 1045.524,A -85,B 0,C 180,E1 6920.975,E2 6920.975} C_VEL
LIN {X 0,Y 627.831,Z 1051.464,A -85,B 0,C 180,E1 6924.46,E2 6924.46} C_VEL
LIN {X 0,Y 627.794,Z 1053.345,A -85,B 0,C 180,E1 6928.617,E2 6928.617} C_VEL
LIN {X 0,Y 627.886,Z 1049.723,A -85,B 0,C 180,E1 6932.767,E2 6932.767} C_VEL
LIN {X 0,Y 628.12,Z 1040.364,A -85,B 0,C 180,E1 6936.929,E2 6936.929} C_VEL
LIN {X 0,Y 628.626,Z 1024.854,A -85,B 0,C 180,E1 6941.12,E2 6941.12} C_VEL
LIN {X 0,Y 629.67,Z 1004.575,A -85,B 0,C 180,E1 6944.995,E2 6944.995} C_VEL
LIN {X 0,Y 631.476,Z 978.997,A -85,B 0,C 180,E1 6948.692,E2 6948.692} C_VEL
LIN {X 0,Y 634.112,Z 946.563,A -85,B 0,C 180,E1 6952.296,E2 6952.296} C_VEL
LIN {X 0,Y 637.267,Z 909.907,A -85,B 0,C 180,E1 6955.438,E2 6955.438} C_VEL
LIN {X 0,Y 640.85,Z 868.972,A -85,B 0,C 180,E1 6958.118,E2 6958.118} C_VEL
LIN {X 0,Y 644.162,Z 824.463,A -85,B 0,C 180,E1 6960.263,E2 6960.263} C_VEL
LIN {X 0,Y 647.014,Z 776.057,A -85,B 0,C 180,E1 6961.839,E2 6961.839} C_VEL
LIN {X 0,Y 647.363,Z 750.803,A -85,B 0,C 180,E1 6962.422,E2 6962.422} C_VEL
LIN {X 0,Y 626.961,Z 707.31,A -85,B 0,C 180,E1 6964.451,E2 6964.451} C_VEL
LIN {X 0,Y 626.929,Z 707.31,A -85,B 0,C 180,E1 6969.328,E2 6969.328} C_VEL
LIN {X 0,Y 626.959,Z 707.31,A -85,B 0,C 180,E1 6975.494,E2 6975.494} C_VEL
LIN {X 0,Y 626.953,Z 707.31,A -85,B 0,C 180,E1 6981.062,E2 6981.062} C_VEL
LIN {X 0,Y 627.005,Z 707.31,A -85,B 0,C 180,E1 6986.226,E2 6986.226} C_VEL
LIN {X 0,Y 627.057,Z 707.31,A -85,B 0,C 180,E1 6991.094,E2 6991.094} C_VEL
LIN {X 0,Y 626.99,Z 707.31,A -85,B 0,C 180,E1 6996.7,E2 6996.7} C_VEL
LIN {X 0,Y 627.049,Z 707.31,A -85,B 0,C 180,E1 7001.687,E2 7001.687} C_VEL
LIN {X 0,Y 627.559,Z 707.31,A -85,B 0,C 180,E1 7007.445,E2 7007.445} C_VEL
LIN {X 0,Y 627.491,Z 707.31,A -85,B 0,C 180,E1 7013.062,E2 7013.062} C_VEL
LIN {X 0,Y 627.205,Z 707.31,A -85,B 0,C 180,E1 7017.228,E2 7017.228} C_VEL
LIN {X 0,Y 627.694,Z 707.31,A -85,B 0,C 180,E1 7021.381,E2 7021.381} C_VEL
LIN {X 0,Y 627.6,Z 707.31,A -85,B 0,C 180,E1 7028.327,E2 7028.327} C_VEL
LIN {X 0,Y 627.259,Z 707.31,A -85,B 0,C 180,E1 7033.978,E2 7033.978} C_VEL
LIN {X 0,Y 627.106,Z 707.31,A -85,B 0,C 180,E1 7039.771,E2 7039.771} C_VEL
LIN {X 0,Y 627.055,Z 707.31,A -85,B 0,C 180,E1 7045.782,E2 7045.782} C_VEL
LIN {X 0,Y 627.088,Z 707.31,A -85,B 0,C 180,E1 7050.493,E2 7050.493} C_VEL
LIN {X 0,Y 627.015,Z 707.31,A -85,B 0,C 180,E1 7055.45,E2 7055.45} C_VEL
LIN {X 0,Y 626.884,Z 707.31,A -85,B 0,C 180,E1 7061.462,E2 7061.462} C_VEL
LIN {X 0,Y 626.872,Z 707.31,A -85,B 0,C 180,E1 7062.507,E2 7062.507} C_VEL
LIN {X 0,Y 622.984,Z 707.31,A -85,B 0,C 180,E1 7064.066,E2 7064.066} C_VEL
LIN {X 0,Y 618.949,Z 707.31,A -85,B 0,C 180,E1 7065.645,E2 7065.645} C_VEL
LIN {X 0,Y 618.949,Z 707.31,A -85,B 0,C 180,E1 7071.574,E2 7071.574} C_VEL
LIN {X 0,Y 619,Z 707.31,A -85,B 0,C 180,E1 7072.599,E2 7072.599} C_VEL
LIN {X 0,Y 642.09,Z 755.488,A -85,B 0,C 180,E1 7074.797,E2 7074.797} C_VEL
LIN {X 0,Y 640.234,Z 805.148,A -85,B 0,C 180,E1 7075.725,E2 7075.725} C_VEL
LIN {X 0,Y 637.217,Z 853.867,A -85,B 0,C 180,E1 7077.322,E2 7077.322} C_VEL
LIN {X 0,Y 633.701,Z 898.602,A -85,B 0,C 180,E1 7079.477,E2 7079.477} C_VEL
LIN {X 0,Y 629.874,Z 941.604,A -85,B 0,C 180,E1 7082.313,E2 7082.313} C_VEL
LIN {X 0,Y 626.512,Z 978.418,A -85,B 0,C 180,E1 7085.53,E2 7085.53} C_VEL
LIN {X 0,Y 623.662,Z 1011.108,A -85,B 0,C 180,E1 7089.263,E2 7089.263} C_VEL
LIN {X 0,Y 621.74,Z 1038.248,A -85,B 0,C 180,E1 7093.357,E2 7093.357} C_VEL
LIN {X 0,Y 620.637,Z 1058.798,A -85,B 0,C 180,E1 7097.585,E2 7097.585} C_VEL
LIN {X 0,Y 620.184,Z 1072.156,A -85,B 0,C 180,E1 7101.569,E2 7101.569} C_VEL
LIN {X 0,Y 620.024,Z 1079.664,A -85,B 0,C 180,E1 7105.092,E2 7105.092} C_VEL
LIN {X 0,Y 619.933,Z 1083.166,A -85,B 0,C 180,E1 7108.599,E2 7108.599} C_VEL
LIN {X 0,Y 620.092,Z 1082.215,A -85,B 0,C 180,E1 7112.801,E2 7112.801} C_VEL
LIN {X 0,Y 620.015,Z 1075.635,A -85,B 0,C 180,E1 7117.019,E2 7117.019} C_VEL
LIN {X 0,Y 620.448,Z 1063.175,A -85,B 0,C 180,E1 7121.267,E2 7121.267} C_VEL
LIN {X 0,Y 621.319,Z 1046.039,A -85,B 0,C 180,E1 7125.2,E2 7125.2} C_VEL
LIN {X 0,Y 622.975,Z 1021.13,A -85,B 0,C 180,E1 7129.355,E2 7129.355} C_VEL
LIN {X 0,Y 625.524,Z 989.642,A -85,B 0,C 180,E1 7133.298,E2 7133.298} C_VEL
LIN {X 0,Y 628.863,Z 952.76,A -85,B 0,C 180,E1 7136.804,E2 7136.804} C_VEL
LIN {X 0,Y 632.561,Z 912.262,A -85,B 0,C 180,E1 7139.709,E2 7139.709} C_VEL
LIN {X 0,Y 636.192,Z 869.03,A -85,B 0,C 180,E1 7142.022,E2 7142.022} C_VEL
LIN {X 0,Y 639.271,Z 823.484,A -85,B 0,C 180,E1 7143.75,E2 7143.75} C_VEL
LIN {X 0,Y 641.458,Z 776.143,A -85,B 0,C 180,E1 7144.891,E2 7144.891} C_VEL
LIN {X 0,Y 641.367,Z 753.601,A -85,B 0,C 180,E1 7145.273,E2 7145.273} C_VEL
LIN {X 0,Y 619.063,Z 707.31,A -85,B 0,C 180,E1 7147.443,E2 7147.443} C_VEL
LIN {X 0,Y 619.013,Z 707.31,A -85,B 0,C 180,E1 7153.271,E2 7153.271} C_VEL
LIN {X 0,Y 618.981,Z 707.31,A -85,B 0,C 180,E1 7159.37,E2 7159.37} C_VEL
LIN {X 0,Y 619.05,Z 707.31,A -85,B 0,C 180,E1 7164.023,E2 7164.023} C_VEL
LIN {X 0,Y 619.127,Z 707.31,A -85,B 0,C 180,E1 7169.072,E2 7169.072} C_VEL
LIN {X 0,Y 619.155,Z 707.31,A -85,B 0,C 180,E1 7173.864,E2 7173.864} C_VEL
LIN {X 0,Y 619.161,Z 707.31,A -85,B 0,C 180,E1 7179.965,E2 7179.965} C_VEL
LIN {X 0,Y 619.344,Z 707.31,A -85,B 0,C 180,E1 7185.84,E2 7185.84} C_VEL
LIN {X 0,Y 619.672,Z 707.31,A -85,B 0,C 180,E1 7191.565,E2 7191.565} C_VEL
LIN {X 0,Y 619.789,Z 707.31,A -85,B 0,C 180,E1 7198.602,E2 7198.602} C_VEL
LIN {X 0,Y 619.509,Z 707.31,A -85,B 0,C 180,E1 7205.618,E2 7205.618} C_VEL
LIN {X 0,Y 619.419,Z 707.31,A -85,B 0,C 180,E1 7211.88,E2 7211.88} C_VEL
LIN {X 0,Y 619.158,Z 707.31,A -85,B 0,C 180,E1 7217.347,E2 7217.347} C_VEL
LIN {X 0,Y 619.268,Z 707.31,A -85,B 0,C 180,E1 7223.052,E2 7223.052} C_VEL
LIN {X 0,Y 618.974,Z 707.31,A -85,B 0,C 180,E1 7228.194,E2 7228.194} C_VEL
LIN {X 0,Y 618.976,Z 707.31,A -85,B 0,C 180,E1 7234.273,E2 7234.273} C_VEL
LIN {X 0,Y 619.029,Z 707.31,A -85,B 0,C 180,E1 7239.533,E2 7239.533} C_VEL
LIN {X 0,Y 619.04,Z 707.31,A -85,B 0,C 180,E1 7245.231,E2 7245.231} C_VEL
LIN {X 0,Y 619.143,Z 708.094,A -85,B 0,C 180,E1 7250.941,E2 7250.941} C_VEL
LIN {X 0,Y 641.339,Z 755.296,A -85,B 0,C 180,E1 7253.208,E2 7253.208} C_VEL
LIN {X 0,Y 639.196,Z 798.806,A -85,B 0,C 180,E1 7254.334,E2 7254.334} C_VEL
LIN {X 0,Y 636.056,Z 842.719,A -85,B 0,C 180,E1 7256.057,E2 7256.057} C_VEL
LIN {X 0,Y 632.414,Z 885.13,A -85,B 0,C 180,E1 7258.39,E2 7258.39} C_VEL
LIN {X 0,Y 628.63,Z 925.33,A -85,B 0,C 180,E1 7261.366,E2 7261.366} C_VEL
LIN {X 0,Y 625.537,Z 960.185,A -85,B 0,C 180,E1 7264.72,E2 7264.72} C_VEL
LIN {X 0,Y 622.957,Z 991.133,A -85,B 0,C 180,E1 7268.6,E2 7268.6} C_VEL
LIN {X 0,Y 621.316,Z 1015.908,A -85,B 0,C 180,E1 7272.729,E2 7272.729} C_VEL
LIN {X 0,Y 620.431,Z 1034.133,A -85,B 0,C 180,E1 7276.943,E2 7276.943} C_VEL
LIN {X 0,Y 620.033,Z 1045.465,A -85,B 0,C 180,E1 7280.86,E2 7280.86} C_VEL
LIN {X 0,Y 619.934,Z 1051.433,A -85,B 0,C 180,E1 7284.389,E2 7284.389} C_VEL
LIN {X 0,Y 619.898,Z 1053.351,A -85,B 0,C 180,E1 7288.6,E2 7288.6} C_VEL
LIN {X 0,Y 619.993,Z 1049.768,A -85,B 0,C 180,E1 7292.803,E2 7292.803} C_VEL
LIN {X 0,Y 620.241,Z 1040.436,A -85,B 0,C 180,E1 7297.018,E2 7297.018} C_VEL
LIN {X 0,Y 620.779,Z 1024.969,A -85,B 0,C 180,E1 7301.262,E2 7301.262} C_VEL
LIN {X 0,Y 622.008,Z 1003.661,A -85,B 0,C 180,E1 7305.365,E2 7305.365} C_VEL
LIN {X 0,Y 623.933,Z 977.329,A -85,B 0,C 180,E1 7309.167,E2 7309.167} C_VEL
LIN {X 0,Y 626.638,Z 946.855,A -85,B 0,C 180,E1 7312.576,E2 7312.576} C_VEL
LIN {X 0,Y 630.204,Z 909.172,A -85,B 0,C 180,E1 7315.839,E2 7315.839} C_VEL
LIN {X 0,Y 633.918,Z 869.187,A -85,B 0,C 180,E1 7318.482,E2 7318.482} C_VEL
LIN {X 0,Y 637.506,Z 823.695,A -85,B 0,C 180,E1 7320.685,E2 7320.685} C_VEL
LIN {X 0,Y 640.398,Z 777.278,A -85,B 0,C 180,E1 7322.207,E2 7322.207} C_VEL
LIN {X 0,Y 640.961,Z 753.911,A -85,B 0,C 180,E1 7322.755,E2 7322.755} C_VEL
LIN {X 0,Y 619.039,Z 707.31,A -85,B 0,C 180,E1 7324.984,E2 7324.984} C_VEL
LIN {X 0,Y 618.991,Z 707.31,A -85,B 0,C 180,E1 7330.627,E2 7330.627} C_VEL
LIN {X 0,Y 619.056,Z 707.31,A -85,B 0,C 180,E1 7336.729,E2 7336.729} C_VEL
LIN {X 0,Y 619.007,Z 707.31,A -85,B 0,C 180,E1 7342.261,E2 7342.261} C_VEL
LIN {X 0,Y 619.11,Z 707.31,A -85,B 0,C 180,E1 7347.416,E2 7347.416} C_VEL
LIN {X 0,Y 619.142,Z 707.31,A -85,B 0,C 180,E1 7352.285,E2 7352.285} C_VEL
LIN {X 0,Y 619.177,Z 707.31,A -85,B 0,C 180,E1 7358.441,E2 7358.441} C_VEL
LIN {X 0,Y 619.296,Z 707.31,A -85,B 0,C 180,E1 7364.383,E2 7364.383} C_VEL
LIN {X 0,Y 619.595,Z 707.31,A -85,B 0,C 180,E1 7368.714,E2 7368.714} C_VEL
LIN {X 0,Y 619.72,Z 707.31,A -85,B 0,C 180,E1 7374.384,E2 7374.384} C_VEL
LIN {X 0,Y 619.801,Z 707.31,A -85,B 0,C 180,E1 7381.398,E2 7381.398} C_VEL
LIN {X 0,Y 619.682,Z 707.31,A -85,B 0,C 180,E1 7388.435,E2 7388.435} C_VEL
LIN {X 0,Y 619.355,Z 707.31,A -85,B 0,C 180,E1 7394.16,E2 7394.16} C_VEL
LIN {X 0,Y 619.168,Z 707.31,A -85,B 0,C 180,E1 7400.035,E2 7400.035} C_VEL
LIN {X 0,Y 619.165,Z 707.31,A -85,B 0,C 180,E1 7406.136,E2 7406.136} C_VEL
LIN {X 0,Y 619.129,Z 707.31,A -85,B 0,C 180,E1 7411.054,E2 7411.054} C_VEL
LIN {X 0,Y 619.054,Z 707.31,A -85,B 0,C 180,E1 7416.116,E2 7416.116} C_VEL
LIN {X 0,Y 618.982,Z 707.31,A -85,B 0,C 180,E1 7421.373,E2 7421.373} C_VEL
LIN {X 0,Y 618.949,Z 707.31,A -85,B 0,C 180,E1 7425.645,E2 7425.645} C_VEL
LIN {X 0,Y 614.941,Z 707.31,A -85,B 0,C 180,E1 7427.214,E2 7427.214} C_VEL
LIN {X 0,Y 610.97,Z 707.31,A -85,B 0,C 180,E1 7428.803,E2 7428.803} C_VEL
LIN {X 0,Y 611.082,Z 708.049,A -85,B 0,C 180,E1 7432.069,E2 7432.069} C_VEL
LIN {X 0,Y 635.58,Z 759.3,A -85,B 0,C 180,E1 7434.447,E2 7434.447} C_VEL
LIN {X 0,Y 633.51,Z 807.302,A -85,B 0,C 180,E1 7435.384,E2 7435.384} C_VEL
LIN {X 0,Y 630.405,Z 854.635,A -85,B 0,C 180,E1 7436.97,E2 7436.97} C_VEL
LIN {X 0,Y 626.578,Z 899.888,A -85,B 0,C 180,E1 7439.189,E2 7439.189} C_VEL
LIN {X 0,Y 622.658,Z 941.388,A -85,B 0,C 180,E1 7441.964,E2 7441.964} C_VEL
LIN {X 0,Y 619.09,Z 978.812,A -85,B 0,C 180,E1 7445.259,E2 7445.259} C_VEL
LIN {X 0,Y 615.994,Z 1011.844,A -85,B 0,C 180,E1 7449.096,E2 7449.096} C_VEL
LIN {X 0,Y 613.964,Z 1038.249,A -85,B 0,C 180,E1 7453.14,E2 7453.14} C_VEL
LIN {X 0,Y 612.784,Z 1059.359,A -85,B 0,C 180,E1 7457.56,E2 7457.56} C_VEL
LIN {X 0,Y 612.284,Z 1073.249,A -85,B 0,C 180,E1 7461.866,E2 7461.866} C_VEL
LIN {X 0,Y 612.091,Z 1080.646,A -85,B 0,C 180,E1 7465.74,E2 7465.74} C_VEL
LIN {X 0,Y 612.132,Z 1083.5,A -85,B 0,C 180,E1 7469.999,E2 7469.999} C_VEL
LIN {X 0,Y 612.158,Z 1080.648,A -85,B 0,C 180,E1 7474.258,E2 7474.258} C_VEL
LIN {X 0,Y 612.257,Z 1072.16,A -85,B 0,C 180,E1 7478.54,E2 7478.54} C_VEL
LIN {X 0,Y 612.775,Z 1059.37,A -85,B 0,C 180,E1 7482.437,E2 7482.437} C_VEL
LIN {X 0,Y 613.868,Z 1038.252,A -85,B 0,C 180,E1 7486.861,E2 7486.861} C_VEL
LIN {X 0,Y 615.903,Z 1012.145,A -85,B 0,C 180,E1 7490.864,E2 7490.864} C_VEL
LIN {X 0,Y 618.848,Z 980.19,A -85,B 0,C 180,E1 7494.6,E2 7494.6} C_VEL
LIN {X 0,Y 622.466,Z 943.747,A -85,B 0,C 180,E1 7497.845,E2 7497.845} C_VEL
LIN {X 0,Y 626.097,Z 905.848,A -85,B 0,C 180,E1 7500.448,E2 7500.448} C_VEL
LIN {X 0,Y 629.63,Z 865.398,A -85,B 0,C 180,E1 7502.561,E2 7502.561} C_VEL
LIN {X 0,Y 632.816,Z 821.371,A -85,B 0,C 180,E1 7504.212,E2 7504.212} C_VEL
LIN {X 0,Y 635.112,Z 773.159,A -85,B 0,C 180,E1 7505.35,E2 7505.35} C_VEL
LIN {X 0,Y 634.803,Z 755.914,A -85,B 0,C 180,E1 7505.657,E2 7505.657} C_VEL
LIN {X 0,Y 611.122,Z 707.31,A -85,B 0,C 180,E1 7508.04,E2 7508.04} C_VEL
LIN {X 0,Y 611.075,Z 707.31,A -85,B 0,C 180,E1 7514.019,E2 7514.019} C_VEL
LIN {X 0,Y 611.074,Z 707.31,A -85,B 0,C 180,E1 7520.242,E2 7520.242} C_VEL
LIN {X 0,Y 611.126,Z 707.31,A -85,B 0,C 180,E1 7525.231,E2 7525.231} C_VEL
LIN {X 0,Y 611.193,Z 707.31,A -85,B 0,C 180,E1 7530.275,E2 7530.275} C_VEL
LIN {X 0,Y 611.17,Z 707.31,A -85,B 0,C 180,E1 7535.073,E2 7535.073} C_VEL
LIN {X 0,Y 611.226,Z 707.31,A -85,B 0,C 180,E1 7540.41,E2 7540.41} C_VEL
LIN {X 0,Y 611.41,Z 707.31,A -85,B 0,C 180,E1 7545.652,E2 7545.652} C_VEL
LIN {X 0,Y 611.683,Z 707.31,A -85,B 0,C 180,E1 7550.016,E2 7550.016} C_VEL
LIN {X 0,Y 611.547,Z 707.31,A -85,B 0,C 180,E1 7554.314,E2 7554.314} C_VEL
LIN {X 0,Y 611.679,Z 707.31,A -85,B 0,C 180,E1 7560.003,E2 7560.003} C_VEL
LIN {X 0,Y 611.58,Z 707.31,A -85,B 0,C 180,E1 7565.691,E2 7565.691} C_VEL
LIN {X 0,Y 611.568,Z 707.31,A -85,B 0,C 180,E1 7571.436,E2 7571.436} C_VEL
LIN {X 0,Y 611.259,Z 707.31,A -85,B 0,C 180,E1 7577.31,E2 7577.31} C_VEL
LIN {X 0,Y 611.388,Z 707.31,A -85,B 0,C 180,E1 7581.829,E2 7581.829} C_VEL
LIN {X 0,Y 611.1,Z 707.31,A -85,B 0,C 180,E1 7586.784,E2 7586.784} C_VEL
LIN {X 0,Y 611.07,Z 707.31,A -85,B 0,C 180,E1 7592.525,E2 7592.525} C_VEL
LIN {X 0,Y 611.079,Z 707.31,A -85,B 0,C 180,E1 7598.317,E2 7598.317} C_VEL
LIN {X 0,Y 611.114,Z 707.31,A -85,B 0,C 180,E1 7604.019,E2 7604.019} C_VEL
LIN {X 0,Y 611.182,Z 707.31,A -85,B 0,C 180,E1 7610.322,E2 7610.322} C_VEL
LIN {X 0,Y 634.729,Z 757.819,A -85,B 0,C 180,E1 7612.842,E2 7612.842} C_VEL
LIN {X 0,Y 632.356,Z 802.447,A -85,B 0,C 180,E1 7614.048,E2 7614.048} C_VEL
LIN {X 0,Y 629.173,Z 844.262,A -85,B 0,C 180,E1 7615.737,E2 7615.737} C_VEL
LIN {X 0,Y 625.33,Z 886.191,A -85,B 0,C 180,E1 7618.083,E2 7618.083} C_VEL
LIN {X 0,Y 621.4,Z 925.496,A -85,B 0,C 180,E1 7621.028,E2 7621.028} C_VEL
LIN {X 0,Y 618.011,Z 960.47,A -85,B 0,C 180,E1 7624.453,E2 7624.453} C_VEL
LIN {X 0,Y 615.258,Z 990.945,A -85,B 0,C 180,E1 7628.319,E2 7628.319} C_VEL
LIN {X 0,Y 613.556,Z 1015.91,A -85,B 0,C 180,E1 7632.532,E2 7632.532} C_VEL
LIN {X 0,Y 612.577,Z 1034.031,A -85,B 0,C 180,E1 7636.773,E2 7636.773} C_VEL
LIN {X 0,Y 612.168,Z 1045.406,A -85,B 0,C 180,E1 7640.741,E2 7640.741} C_VEL
LIN {X 0,Y 612.03,Z 1051.4,A -85,B 0,C 180,E1 7644.317,E2 7644.317} C_VEL
LIN {X 0,Y 611.996,Z 1053.358,A -85,B 0,C 180,E1 7648.582,E2 7648.582} C_VEL
LIN {X 0,Y 612.096,Z 1049.813,A -85,B 0,C 180,E1 7652.839,E2 7652.839} C_VEL
LIN {X 0,Y 612.359,Z 1040.508,A -85,B 0,C 180,E1 7657.108,E2 7657.108} C_VEL
LIN {X 0,Y 612.93,Z 1025.083,A -85,B 0,C 180,E1 7661.408,E2 7661.408} C_VEL
LIN {X 0,Y 614.264,Z 1003.823,A -85,B 0,C 180,E1 7665.563,E2 7665.563} C_VEL
LIN {X 0,Y 616.3,Z 977.751,A -85,B 0,C 180,E1 7669.388,E2 7669.388} C_VEL
LIN {X 0,Y 619.202,Z 947.163,A -85,B 0,C 180,E1 7672.863,E2 7672.863} C_VEL
LIN {X 0,Y 623.057,Z 909.758,A -85,B 0,C 180,E1 7676.158,E2 7676.158} C_VEL
LIN {X 0,Y 627.113,Z 868.53,A -85,B 0,C 180,E1 7678.901,E2 7678.901} C_VEL
LIN {X 0,Y 630.811,Z 824.125,A -85,B 0,C 180,E1 7681.067,E2 7681.067} C_VEL
LIN {X 0,Y 633.87,Z 777.589,A -85,B 0,C 180,E1 7682.607,E2 7682.607} C_VEL
LIN {X 0,Y 634.451,Z 756.611,A -85,B 0,C 180,E1 7683.111,E2 7683.111} C_VEL
LIN {X 0,Y 611.1,Z 707.31,A -85,B 0,C 180,E1 7685.591,E2 7685.591} C_VEL
LIN {X 0,Y 611.073,Z 707.31,A -85,B 0,C 180,E1 7690.15,E2 7690.15} C_VEL
LIN {X 0,Y 611.124,Z 707.31,A -85,B 0,C 180,E1 7696.025,E2 7696.025} C_VEL
LIN {X 0,Y 611.1,Z 707.31,A -85,B 0,C 180,E1 7701.685,E2 7701.685} C_VEL
LIN {X 0,Y 611.214,Z 707.31,A -85,B 0,C 180,E1 7707.456,E2 7707.456} C_VEL
LIN {X 0,Y 611.222,Z 707.31,A -85,B 0,C 180,E1 7713.493,E2 7713.493} C_VEL
LIN {X 0,Y 611.256,Z 707.31,A -85,B 0,C 180,E1 7719.689,E2 7719.689} C_VEL
LIN {X 0,Y 611.558,Z 707.31,A -85,B 0,C 180,E1 7725.651,E2 7725.651} C_VEL
LIN {X 0,Y 611.735,Z 707.31,A -85,B 0,C 180,E1 7731.45,E2 7731.45} C_VEL
LIN {X 0,Y 611.721,Z 707.31,A -85,B 0,C 180,E1 7735.735,E2 7735.735} C_VEL
LIN {X 0,Y 611.887,Z 707.31,A -85,B 0,C 180,E1 7741.417,E2 7741.417} C_VEL
LIN {X 0,Y 611.772,Z 707.31,A -85,B 0,C 180,E1 7747.763,E2 7747.763} C_VEL
LIN {X 0,Y 611.534,Z 707.31,A -85,B 0,C 180,E1 7752.884,E2 7752.884} C_VEL
LIN {X 0,Y 611.229,Z 707.31,A -85,B 0,C 180,E1 7758.799,E2 7758.799} C_VEL
LIN {X 0,Y 611.133,Z 707.31,A -85,B 0,C 180,E1 7763.439,E2 7763.439} C_VEL
LIN {X 0,Y 611.243,Z 707.31,A -85,B 0,C 180,E1 7768.099,E2 7768.099} C_VEL
LIN {X 0,Y 611.207,Z 707.31,A -85,B 0,C 180,E1 7773.052,E2 7773.052} C_VEL
LIN {X 0,Y 611.101,Z 707.31,A -85,B 0,C 180,E1 7778.308,E2 7778.308} C_VEL
LIN {X 0,Y 611.057,Z 707.31,A -85,B 0,C 180,E1 7784.012,E2 7784.012} C_VEL
LIN {X 0,Y 610.97,Z 707.31,A -85,B 0,C 180,E1 7788.803,E2 7788.803} C_VEL
LIN {X 0,Y 606.987,Z 707.31,A -85,B 0,C 180,E1 7789.839,E2 7789.839} C_VEL
LIN {X 0,Y 603.091,Z 707.31,A -85,B 0,C 180,E1 7790.889,E2 7790.889} C_VEL
LIN {X 0,Y 603.132,Z 707.522,A -85,B 0,C 180,E1 7791.488,E2 7791.488} C_VEL
LIN {X 0,Y 629.105,Z 761.329,A -85,B 0,C 180,E1 7794.062,E2 7794.062} C_VEL
LIN {X 0,Y 626.91,Z 808.107,A -85,B 0,C 180,E1 7795,E2 7795} C_VEL
LIN {X 0,Y 623.63,Z 855.003,A -85,B 0,C 180,E1 7796.593,E2 7796.593} C_VEL
LIN {X 0,Y 619.69,Z 899.28,A -85,B 0,C 180,E1 7798.783,E2 7798.783} C_VEL
LIN {X 0,Y 615.543,Z 940.748,A -85,B 0,C 180,E1 7801.574,E2 7801.574} C_VEL
LIN {X 0,Y 611.679,Z 978.61,A -85,B 0,C 180,E1 7804.939,E2 7804.939} C_VEL
LIN {X 0,Y 608.513,Z 1011.178,A -85,B 0,C 180,E1 7808.732,E2 7808.732} C_VEL
LIN {X 0,Y 606.204,Z 1038.25,A -85,B 0,C 180,E1 7812.918,E2 7812.918} C_VEL
LIN {X 0,Y 604.946,Z 1059.387,A -85,B 0,C 180,E1 7817.404,E2 7817.404} C_VEL
LIN {X 0,Y 604.381,Z 1073.776,A -85,B 0,C 180,E1 7821.957,E2 7821.957} C_VEL
LIN {X 0,Y 604.191,Z 1080.645,A -85,B 0,C 180,E1 7825.684,E2 7825.684} C_VEL
LIN {X 0,Y 604.248,Z 1083.5,A -85,B 0,C 180,E1 7829.999,E2 7829.999} C_VEL
LIN {X 0,Y 604.253,Z 1080.648,A -85,B 0,C 180,E1 7834.314,E2 7834.314} C_VEL
LIN {X 0,Y 604.31,Z 1073.411,A -85,B 0,C 180,E1 7838.181,E2 7838.181} C_VEL
LIN {X 0,Y 604.899,Z 1059.376,A -85,B 0,C 180,E1 7842.6,E2 7842.6} C_VEL
LIN {X 0,Y 605.999,Z 1040.213,A -85,B 0,C 180,E1 7846.712,E2 7846.712} C_VEL
LIN {X 0,Y 607.898,Z 1016.12,A -85,B 0,C 180,E1 7850.58,E2 7850.58} C_VEL
LIN {X 0,Y 610.752,Z 987.084,A -85,B 0,C 180,E1 7854.166,E2 7854.166} C_VEL
LIN {X 0,Y 614.415,Z 951.452,A -85,B 0,C 180,E1 7857.561,E2 7857.561} C_VEL
LIN {X 0,Y 618.549,Z 911.818,A -85,B 0,C 180,E1 7860.452,E2 7860.452} C_VEL
LIN {X 0,Y 622.624,Z 867.915,A -85,B 0,C 180,E1 7862.841,E2 7862.841} C_VEL
LIN {X 0,Y 626.207,Z 821.408,A -85,B 0,C 180,E1 7864.614,E2 7864.614} C_VEL
LIN {X 0,Y 628.687,Z 772.958,A -85,B 0,C 180,E1 7865.767,E2 7865.767} C_VEL
LIN {X 0,Y 628.271,Z 758.44,A -85,B 0,C 180,E1 7866.041,E2 7866.041} C_VEL
LIN {X 0,Y 604.581,Z 711.771,A -85,B 0,C 180,E1 7868.414,E2 7868.414} C_VEL
LIN {X 0,Y 603.195,Z 707.31,A -85,B 0,C 180,E1 7868.67,E2 7868.67} C_VEL
LIN {X 0,Y 603.105,Z 707.31,A -85,B 0,C 180,E1 7874.711,E2 7874.711} C_VEL
LIN {X 0,Y 603.142,Z 707.31,A -85,B 0,C 180,E1 7881.157,E2 7881.157} C_VEL
LIN {X 0,Y 603.23,Z 707.31,A -85,B 0,C 180,E1 7886.453,E2 7886.453} C_VEL
LIN {X 0,Y 603.309,Z 707.31,A -85,B 0,C 180,E1 7891.537,E2 7891.537} C_VEL
LIN {X 0,Y 603.223,Z 707.31,A -85,B 0,C 180,E1 7896.303,E2 7896.303} C_VEL
LIN {X 0,Y 603.337,Z 707.31,A -85,B 0,C 180,E1 7900.945,E2 7900.945} C_VEL
LIN {X 0,Y 603.594,Z 707.31,A -85,B 0,C 180,E1 7906.944,E2 7906.944} C_VEL
LIN {X 0,Y 603.889,Z 707.31,A -85,B 0,C 180,E1 7912.795,E2 7912.795} C_VEL
LIN {X 0,Y 603.968,Z 707.31,A -85,B 0,C 180,E1 7918.565,E2 7918.565} C_VEL
LIN {X 0,Y 603.716,Z 707.31,A -85,B 0,C 180,E1 7924.321,E2 7924.321} C_VEL
LIN {X 0,Y 603.568,Z 707.31,A -85,B 0,C 180,E1 7930.125,E2 7930.125} C_VEL
LIN {X 0,Y 603.472,Z 707.31,A -85,B 0,C 180,E1 7934.546,E2 7934.546} C_VEL
LIN {X 0,Y 603.412,Z 707.31,A -85,B 0,C 180,E1 7940.587,E2 7940.587} C_VEL
LIN {X 0,Y 603.278,Z 707.31,A -85,B 0,C 180,E1 7945.282,E2 7945.282} C_VEL
LIN {X 0,Y 603.137,Z 707.31,A -85,B 0,C 180,E1 7951.323,E2 7951.323} C_VEL
LIN {X 0,Y 603.136,Z 707.31,A -85,B 0,C 180,E1 7957.088,E2 7957.088} C_VEL
LIN {X 0,Y 603.158,Z 707.31,A -85,B 0,C 180,E1 7963.231,E2 7963.231} C_VEL
LIN {X 0,Y 603.204,Z 707.31,A -85,B 0,C 180,E1 7969.557,E2 7969.557} C_VEL
LIN {X 0,Y 603.238,Z 707.519,A -85,B 0,C 180,E1 7969.752,E2 7969.752} C_VEL
LIN {X 0,Y 627.045,Z 757.613,A -85,B 0,C 180,E1 7972.336,E2 7972.336} C_VEL
LIN {X 0,Y 628.066,Z 764.586,A -85,B 0,C 180,E1 7972.576,E2 7972.576} C_VEL
LIN {X 0,Y 625.237,Z 810.138,A -85,B 0,C 180,E1 7973.896,E2 7973.896} C_VEL
LIN {X 0,Y 621.394,Z 855.397,A -85,B 0,C 180,E1 7975.883,E2 7975.883} C_VEL
LIN {X 0,Y 617.24,Z 897.917,A -85,B 0,C 180,E1 7978.496,E2 7978.496} C_VEL
LIN {X 0,Y 613.03,Z 936.151,A -85,B 0,C 180,E1 7981.623,E2 7981.623} C_VEL
LIN {X 0,Y 609.487,Z 969.759,A -85,B 0,C 180,E1 7985.229,E2 7985.229} C_VEL
LIN {X 0,Y 606.923,Z 998.872,A -85,B 0,C 180,E1 7989.285,E2 7989.285} C_VEL
LIN {X 0,Y 605.22,Z 1022.131,A -85,B 0,C 180,E1 7993.64,E2 7993.64} C_VEL
LIN {X 0,Y 604.549,Z 1038.042,A -85,B 0,C 180,E1 7997.858,E2 7997.858} C_VEL
LIN {X 0,Y 604.238,Z 1047.944,A -85,B 0,C 180,E1 8001.891,E2 8001.891} C_VEL
LIN {X 0,Y 604.135,Z 1052.648,A -85,B 0,C 180,E1 8005.685,E2 8005.685} C_VEL
LIN {X 0,Y 604.324,Z 1052.808,A -85,B 0,C 180,E1 8010.001,E2 8010.001} C_VEL
LIN {X 0,Y 604.274,Z 1047.443,A -85,B 0,C 180,E1 8014.315,E2 8014.315} C_VEL
LIN {X 0,Y 604.517,Z 1036.157,A -85,B 0,C 180,E1 8018.651,E2 8018.651} C_VEL
LIN {X 0,Y 605.349,Z 1020.279,A -85,B 0,C 180,E1 8022.662,E2 8022.662} C_VEL
LIN {X 0,Y 606.94,Z 998.477,A -85,B 0,C 180,E1 8026.687,E2 8026.687} C_VEL
LIN {X 0,Y 609.454,Z 970.339,A -85,B 0,C 180,E1 8030.612,E2 8030.612} C_VEL
LIN {X 0,Y 613.133,Z 935.516,A -85,B 0,C 180,E1 8034.341,E2 8034.341} C_VEL
LIN {X 0,Y 617.389,Z 896.596,A -85,B 0,C 180,E1 8037.501,E2 8037.501} C_VEL
LIN {X 0,Y 621.679,Z 853.976,A -85,B 0,C 180,E1 8040.088,E2 8040.088} C_VEL
LIN {X 0,Y 625.299,Z 810.84,A -85,B 0,C 180,E1 8041.978,E2 8041.978} C_VEL
LIN {X 0,Y 628.039,Z 766.917,A -85,B 0,C 180,E1 8043.271,E2 8043.271} C_VEL
LIN {X 0,Y 627.494,Z 758.242,A -85,B 0,C 180,E1 8043.529,E2 8043.529} C_VEL
LIN {X 0,Y 603.306,Z 708.741,A -85,B 0,C 180,E1 8046.063,E2 8046.063} C_VEL
LIN {X 0,Y 603.18,Z 707.31,A -85,B 0,C 180,E1 8046.101,E2 8046.101} C_VEL
LIN {X 0,Y 603.087,Z 707.31,A -85,B 0,C 180,E1 8051.074,E2 8051.074} C_VEL
LIN {X 0,Y 603.168,Z 707.31,A -85,B 0,C 180,E1 8056.77,E2 8056.77} C_VEL
LIN {X 0,Y 603.175,Z 707.31,A -85,B 0,C 180,E1 8062.914,E2 8062.914} C_VEL
LIN {X 0,Y 603.319,Z 707.31,A -85,B 0,C 180,E1 8068.651,E2 8068.651} C_VEL
LIN {X 0,Y 603.293,Z 707.31,A -85,B 0,C 180,E1 8074.727,E2 8074.727} C_VEL
LIN {X 0,Y 603.325,Z 707.31,A -85,B 0,C 180,E1 8079.41,E2 8079.41} C_VEL
LIN {X 0,Y 603.639,Z 707.31,A -85,B 0,C 180,E1 8085.458,E2 8085.458} C_VEL
LIN {X 0,Y 603.78,Z 707.31,A -85,B 0,C 180,E1 8089.879,E2 8089.879} C_VEL
LIN {X 0,Y 603.818,Z 707.31,A -85,B 0,C 180,E1 8095.68,E2 8095.68} C_VEL
LIN {X 0,Y 603.976,Z 707.31,A -85,B 0,C 180,E1 8101.435,E2 8101.435} C_VEL
LIN {X 0,Y 603.9,Z 707.31,A -85,B 0,C 180,E1 8107.205,E2 8107.205} C_VEL
LIN {X 0,Y 603.607,Z 707.31,A -85,B 0,C 180,E1 8113.056,E2 8113.056} C_VEL
LIN {X 0,Y 603.343,Z 707.31,A -85,B 0,C 180,E1 8119.054,E2 8119.054} C_VEL
LIN {X 0,Y 603.233,Z 707.31,A -85,B 0,C 180,E1 8123.696,E2 8123.696} C_VEL
LIN {X 0,Y 603.29,Z 707.31,A -85,B 0,C 180,E1 8128.503,E2 8128.503} C_VEL
LIN {X 0,Y 603.213,Z 707.31,A -85,B 0,C 180,E1 8134,E2 8134} C_VEL
LIN {X 0,Y 603.152,Z 707.31,A -85,B 0,C 180,E1 8138.907,E2 8138.907} C_VEL
LIN {X 0,Y 603.097,Z 707.31,A -85,B 0,C 180,E1 8145.286,E2 8145.286} C_VEL
LIN {X 0,Y 603.091,Z 707.31,A -85,B 0,C 180,E1 8150.889,E2 8150.889} C_VEL
LIN {X 0,Y 604.077,Z 710.43,A -85,B 0,C 180,E1 8151.451,E2 8151.451} C_VEL
LIN {X 0,Y 606.15,Z 718.751,A -85,B 0,C 180,E1 8151.872,E2 8151.872} C_VEL
LIN {X 0,Y 610.272,Z 737.543,A -85,B 0,C 180,E1 8152.438,E2 8152.438} C_VEL
LIN {X 0,Y 622.616,Z 763.379,A -85,B 0,C 180,E1 8153.669,E2 8153.669} C_VEL
LIN {X 0,Y 620.361,Z 808.58,A -85,B 0,C 180,E1 8154.599,E2 8154.599} C_VEL
LIN {X 0,Y 616.997,Z 854.353,A -85,B 0,C 180,E1 8156.164,E2 8156.164} C_VEL
LIN {X 0,Y 612.706,Z 899.584,A -85,B 0,C 180,E1 8158.421,E2 8158.421} C_VEL
LIN {X 0,Y 608.331,Z 941.076,A -85,B 0,C 180,E1 8161.253,E2 8161.253} C_VEL
LIN {X 0,Y 604.22,Z 978.624,A -85,B 0,C 180,E1 8164.634,E2 8164.634} C_VEL
LIN {X 0,Y 600.879,Z 1011.281,A -85,B 0,C 180,E1 8168.473,E2 8168.473} C_VEL
LIN {X 0,Y 598.46,Z 1038.251,A -85,B 0,C 180,E1 8172.69,E2 8172.69} C_VEL
LIN {X 0,Y 597.108,Z 1059.109,A -85,B 0,C 180,E1 8177.164,E2 8177.164} C_VEL
LIN {X 0,Y 596.547,Z 1072.156,A -85,B 0,C 180,E1 8181.232,E2 8181.232} C_VEL
LIN {X 0,Y 596.338,Z 1079.665,A -85,B 0,C 180,E1 8184.897,E2 8184.897} C_VEL
LIN {X 0,Y 596.245,Z 1083.165,A -85,B 0,C 180,E1 8188.543,E2 8188.543} C_VEL
LIN {X 0,Y 596.4,Z 1082.214,A -85,B 0,C 180,E1 8192.912,E2 8192.912} C_VEL
LIN {X 0,Y 596.376,Z 1075.635,A -85,B 0,C 180,E1 8197.299,E2 8197.299} C_VEL
LIN {X 0,Y 596.902,Z 1063.173,A -85,B 0,C 180,E1 8201.718,E2 8201.718} C_VEL
LIN {X 0,Y 597.97,Z 1045.919,A -85,B 0,C 180,E1 8205.834,E2 8205.834} C_VEL
LIN {X 0,Y 599.867,Z 1021.135,A -85,B 0,C 180,E1 8210.132,E2 8210.132} C_VEL
LIN {X 0,Y 602.946,Z 990.332,A -85,B 0,C 180,E1 8214.105,E2 8214.105} C_VEL
LIN {X 0,Y 606.924,Z 953.84,A -85,B 0,C 180,E1 8217.698,E2 8217.698} C_VEL
LIN {X 0,Y 611.408,Z 913.066,A -85,B 0,C 180,E1 8220.743,E2 8220.743} C_VEL
LIN {X 0,Y 615.646,Z 870.15,A -85,B 0,C 180,E1 8223.127,E2 8223.127} C_VEL
LIN {X 0,Y 619.25,Z 826.168,A -85,B 0,C 180,E1 8224.871,E2 8224.871} C_VEL
LIN {X 0,Y 621.836,Z 781.377,A -85,B 0,C 180,E1 8226.037,E2 8226.037} C_VEL
LIN {X 0,Y 621.985,Z 761.416,A -85,B 0,C 180,E1 8226.415,E2 8226.415} C_VEL
LIN {X 0,Y 597.064,Z 712.273,A -85,B 0,C 180,E1 8228.991,E2 8228.991} C_VEL
LIN {X 0,Y 595.246,Z 707.31,A -85,B 0,C 180,E1 8229.232,E2 8229.232} C_VEL
LIN {X 0,Y 595.186,Z 707.31,A -85,B 0,C 180,E1 8234.533,E2 8234.533} C_VEL
LIN {X 0,Y 595.149,Z 707.31,A -85,B 0,C 180,E1 8240.468,E2 8240.468} C_VEL
LIN {X 0,Y 595.306,Z 707.31,A -85,B 0,C 180,E1 8245.946,E2 8245.946} C_VEL
LIN {X 0,Y 595.354,Z 707.31,A -85,B 0,C 180,E1 8251.081,E2 8251.081} C_VEL
LIN {X 0,Y 595.32,Z 707.31,A -85,B 0,C 180,E1 8256.402,E2 8256.402} C_VEL
LIN {X 0,Y 595.392,Z 707.31,A -85,B 0,C 180,E1 8262.219,E2 8262.219} C_VEL
LIN {X 0,Y 595.813,Z 707.31,A -85,B 0,C 180,E1 8268.263,E2 8268.263} C_VEL
LIN {X 0,Y 595.979,Z 707.31,A -85,B 0,C 180,E1 8272.699,E2 8272.699} C_VEL
LIN {X 0,Y 596.056,Z 707.31,A -85,B 0,C 180,E1 8278.546,E2 8278.546} C_VEL
LIN {X 0,Y 595.806,Z 707.31,A -85,B 0,C 180,E1 8284.379,E2 8284.379} C_VEL
LIN {X 0,Y 595.69,Z 707.31,A -85,B 0,C 180,E1 8290.26,E2 8290.26} C_VEL
LIN {X 0,Y 595.544,Z 707.31,A -85,B 0,C 180,E1 8294.778,E2 8294.778} C_VEL
LIN {X 0,Y 595.508,Z 707.31,A -85,B 0,C 180,E1 8300.873,E2 8300.873} C_VEL
LIN {X 0,Y 595.318,Z 707.31,A -85,B 0,C 180,E1 8305.644,E2 8305.644} C_VEL
LIN {X 0,Y 595.223,Z 707.31,A -85,B 0,C 180,E1 8310.612,E2 8310.612} C_VEL
LIN {X 0,Y 595.22,Z 707.31,A -85,B 0,C 180,E1 8315.846,E2 8315.846} C_VEL
LIN {X 0,Y 595.217,Z 707.31,A -85,B 0,C 180,E1 8321.452,E2 8321.452} C_VEL
LIN {X 0,Y 595.217,Z 707.31,A -85,B 0,C 180,E1 8326.576,E2 8326.576} C_VEL
LIN {X 0,Y 595.297,Z 708.031,A -85,B 0,C 180,E1 8329.136,E2 8329.136} C_VEL
LIN {X 0,Y 618.516,Z 755.308,A -85,B 0,C 180,E1 8331.704,E2 8331.704} C_VEL
LIN {X 0,Y 621.642,Z 764.695,A -85,B 0,C 180,E1 8332.149,E2 8332.149} C_VEL
LIN {X 0,Y 618.68,Z 810.516,A -85,B 0,C 180,E1 8333.491,E2 8333.491} C_VEL
LIN {X 0,Y 614.508,Z 856.747,A -85,B 0,C 180,E1 8335.549,E2 8335.549} C_VEL
LIN {X 0,Y 610.253,Z 898.247,A -85,B 0,C 180,E1 8338.134,E2 8338.134} C_VEL
LIN {X 0,Y 605.644,Z 937.664,A -85,B 0,C 180,E1 8341.408,E2 8341.408} C_VEL
LIN {X 0,Y 601.839,Z 971.591,A -85,B 0,C 180,E1 8345.131,E2 8345.131} C_VEL
LIN {X 0,Y 599.029,Z 1001.048,A -85,B 0,C 180,E1 8349.398,E2 8349.398} C_VEL
LIN {X 0,Y 597.468,Z 1021.997,A -85,B 0,C 180,E1 8353.421,E2 8353.421} C_VEL
LIN {X 0,Y 596.672,Z 1037.955,A -85,B 0,C 180,E1 8357.696,E2 8357.696} C_VEL
LIN {X 0,Y 596.349,Z 1046.861,A -85,B 0,C 180,E1 8361.231,E2 8361.231} C_VEL
LIN {X 0,Y 596.228,Z 1052.628,A -85,B 0,C 180,E1 8365.628,E2 8365.628} C_VEL
LIN {X 0,Y 596.422,Z 1052.826,A -85,B 0,C 180,E1 8370.001,E2 8370.001} C_VEL
LIN {X 0,Y 596.374,Z 1047.491,A -85,B 0,C 180,E1 8374.373,E2 8374.373} C_VEL
LIN {X 0,Y 596.665,Z 1036.242,A -85,B 0,C 180,E1 8378.766,E2 8378.766} C_VEL
LIN {X 0,Y 597.546,Z 1020.03,A -85,B 0,C 180,E1 8382.912,E2 8382.912} C_VEL
LIN {X 0,Y 599.215,Z 998.658,A -85,B 0,C 180,E1 8386.908,E2 8386.908} C_VEL
LIN {X 0,Y 602.056,Z 969.408,A -85,B 0,C 180,E1 8391.047,E2 8391.047} C_VEL
LIN {X 0,Y 605.95,Z 935.303,A -85,B 0,C 180,E1 8394.719,E2 8394.719} C_VEL
LIN {X 0,Y 610.368,Z 897.217,A -85,B 0,C 180,E1 8397.845,E2 8397.845} C_VEL
LIN {X 0,Y 614.807,Z 855.326,A -85,B 0,C 180,E1 8400.427,E2 8400.427} C_VEL
LIN {X 0,Y 618.661,Z 811.757,A -85,B 0,C 180,E1 8402.363,E2 8402.363} C_VEL
LIN {X 0,Y 621.417,Z 769.549,A -85,B 0,C 180,E1 8403.637,E2 8403.637} C_VEL
LIN {X 0,Y 621.188,Z 761.433,A -85,B 0,C 180,E1 8403.873,E2 8403.873} C_VEL
LIN {X 0,Y 598.989,Z 716.166,A -85,B 0,C 180,E1 8406.272,E2 8406.272} C_VEL
LIN {X 0,Y 595.275,Z 707.31,A -85,B 0,C 180,E1 8406.7,E2 8406.7} C_VEL
LIN {X 0,Y 595.163,Z 707.31,A -85,B 0,C 180,E1 8412.402,E2 8412.402} C_VEL
LIN {X 0,Y 595.235,Z 707.31,A -85,B 0,C 180,E1 8417.588,E2 8417.588} C_VEL
LIN {X 0,Y 595.215,Z 707.31,A -85,B 0,C 180,E1 8422.333,E2 8422.333} C_VEL
LIN {X 0,Y 595.314,Z 707.31,A -85,B 0,C 180,E1 8427.683,E2 8427.683} C_VEL
LIN {X 0,Y 595.413,Z 707.31,A -85,B 0,C 180,E1 8432.974,E2 8432.974} C_VEL
LIN {X 0,Y 595.411,Z 707.31,A -85,B 0,C 180,E1 8439.123,E2 8439.123} C_VEL
LIN {X 0,Y 595.699,Z 707.31,A -85,B 0,C 180,E1 8445.26,E2 8445.26} C_VEL
LIN {X 0,Y 595.886,Z 707.31,A -85,B 0,C 180,E1 8449.743,E2 8449.743} C_VEL
LIN {X 0,Y 595.916,Z 707.31,A -85,B 0,C 180,E1 8455.622,E2 8455.622} C_VEL
LIN {X 0,Y 596.063,Z 707.31,A -85,B 0,C 180,E1 8461.454,E2 8461.454} C_VEL
LIN {X 0,Y 595.988,Z 707.31,A -85,B 0,C 180,E1 8467.409,E2 8467.409} C_VEL
LIN {X 0,Y 595.676,Z 707.31,A -85,B 0,C 180,E1 8473.233,E2 8473.233} C_VEL
LIN {X 0,Y 595.406,Z 707.31,A -85,B 0,C 180,E1 8479.319,E2 8479.319} C_VEL
LIN {X 0,Y 595.317,Z 707.31,A -85,B 0,C 180,E1 8484.031,E2 8484.031} C_VEL
LIN {X 0,Y 595.34,Z 707.31,A -85,B 0,C 180,E1 8488.919,E2 8488.919} C_VEL
LIN {X 0,Y 595.307,Z 707.31,A -85,B 0,C 180,E1 8494.054,E2 8494.054} C_VEL
LIN {X 0,Y 595.162,Z 707.31,A -85,B 0,C 180,E1 8500.193,E2 8500.193} C_VEL
LIN {X 0,Y 595.175,Z 707.31,A -85,B 0,C 180,E1 8505.468,E2 8505.468} C_VEL
LIN {X 0,Y 595.24,Z 707.919,A -85,B 0,C 180,E1 8510.905,E2 8510.905} C_VEL
LIN {X 0,Y 610.272,Z 737.543,A -85,B 0,C 180,E1 8512.438,E2 8512.438} C_VEL
LIN {X 0,Y 614.959,Z 753.523,A -85,B 0,C 180,E1 8512.991,E2 8512.991} C_VEL
LIN {X 0,Y 616.04,Z 770.795,A -85,B 0,C 180,E1 8513.355,E2 8513.355} C_VEL
LIN {X 0,Y 613.153,Z 819.739,A -85,B 0,C 180,E1 8514.498,E2 8514.498} C_VEL
LIN {X 0,Y 609.119,Z 866.967,A -85,B 0,C 180,E1 8516.308,E2 8516.308} C_VEL
LIN {X 0,Y 604.485,Z 912.114,A -85,B 0,C 180,E1 8518.81,E2 8518.81} C_VEL
LIN {X 0,Y 599.76,Z 952.923,A -85,B 0,C 180,E1 8521.874,E2 8521.874} C_VEL
LIN {X 0,Y 595.518,Z 990.111,A -85,B 0,C 180,E1 8525.574,E2 8525.574} C_VEL
LIN {X 0,Y 592.239,Z 1020.953,A -85,B 0,C 180,E1 8529.596,E2 8529.596} C_VEL
LIN {X 0,Y 590.123,Z 1045.708,A -85,B 0,C 180,E1 8533.906,E2 8533.906} C_VEL
LIN {X 0,Y 588.964,Z 1064.504,A -85,B 0,C 180,E1 8538.497,E2 8538.497} C_VEL
LIN {X 0,Y 588.536,Z 1075.632,A -85,B 0,C 180,E1 8542.602,E2 8542.602} C_VEL
LIN {X 0,Y 588.4,Z 1080.645,A -85,B 0,C 180,E1 8545.568,E2 8545.568} C_VEL
LIN {X 0,Y 588.464,Z 1083.5,A -85,B 0,C 180,E1 8549.999,E2 8549.999} C_VEL
LIN {X 0,Y 588.447,Z 1080.647,A -85,B 0,C 180,E1 8554.43,E2 8554.43} C_VEL
LIN {X 0,Y 588.534,Z 1073.495,A -85,B 0,C 180,E1 8558.37,E2 8558.37} C_VEL
LIN {X 0,Y 589.17,Z 1060.155,A -85,B 0,C 180,E1 8562.724,E2 8562.724} C_VEL
LIN {X 0,Y 590.354,Z 1042.16,A -85,B 0,C 180,E1 8566.784,E2 8566.784} C_VEL
LIN {X 0,Y 592.297,Z 1019.651,A -85,B 0,C 180,E1 8570.596,E2 8570.596} C_VEL
LIN {X 0,Y 595.66,Z 988.41,A -85,B 0,C 180,E1 8574.619,E2 8574.619} C_VEL
LIN {X 0,Y 599.812,Z 952.91,A -85,B 0,C 180,E1 8578.122,E2 8578.122} C_VEL
LIN {X 0,Y 604.545,Z 911.779,A -85,B 0,C 180,E1 8581.208,E2 8581.208} C_VEL
LIN {X 0,Y 609.152,Z 868.023,A -85,B 0,C 180,E1 8583.635,E2 8583.635} C_VEL
LIN {X 0,Y 613.082,Z 822.178,A -85,B 0,C 180,E1 8585.425,E2 8585.425} C_VEL
LIN {X 0,Y 615.813,Z 775.029,A -85,B 0,C 180,E1 8586.59,E2 8586.59} C_VEL
LIN {X 0,Y 615.564,Z 764.098,A -85,B 0,C 180,E1 8586.816,E2 8586.816} C_VEL
LIN {X 0,Y 592.16,Z 717.646,A -85,B 0,C 180,E1 8589.3,E2 8589.3} C_VEL
LIN {X 0,Y 587.302,Z 707.31,A -85,B 0,C 180,E1 8589.937,E2 8589.937} C_VEL
LIN {X 0,Y 587.266,Z 707.31,A -85,B 0,C 180,E1 8595.84,E2 8595.84} C_VEL
LIN {X 0,Y 587.25,Z 707.31,A -85,B 0,C 180,E1 8601.737,E2 8601.737} C_VEL
LIN {X 0,Y 587.425,Z 707.31,A -85,B 0,C 180,E1 8607.201,E2 8607.201} C_VEL
LIN {X 0,Y 587.45,Z 707.31,A -85,B 0,C 180,E1 8612.336,E2 8612.336} C_VEL
LIN {X 0,Y 587.391,Z 707.31,A -85,B 0,C 180,E1 8618.24,E2 8618.24} C_VEL
LIN {X 0,Y 587.532,Z 707.31,A -85,B 0,C 180,E1 8623.521,E2 8623.521} C_VEL
LIN {X 0,Y 587.943,Z 707.31,A -85,B 0,C 180,E1 8629.609,E2 8629.609} C_VEL
LIN {X 0,Y 587.87,Z 707.31,A -85,B 0,C 180,E1 8634.084,E2 8634.084} C_VEL
LIN {X 0,Y 587.987,Z 707.31,A -85,B 0,C 180,E1 8640.003,E2 8640.003} C_VEL
LIN {X 0,Y 587.816,Z 707.31,A -85,B 0,C 180,E1 8645.922,E2 8645.922} C_VEL
LIN {X 0,Y 587.85,Z 707.31,A -85,B 0,C 180,E1 8651.904,E2 8651.904} C_VEL
LIN {X 0,Y 587.515,Z 707.31,A -85,B 0,C 180,E1 8658.033,E2 8658.033} C_VEL
LIN {X 0,Y 587.581,Z 707.31,A -85,B 0,C 180,E1 8662.762,E2 8662.762} C_VEL
LIN {X 0,Y 587.276,Z 707.31,A -85,B 0,C 180,E1 8668.679,E2 8668.679} C_VEL
LIN {X 0,Y 587.279,Z 707.31,A -85,B 0,C 180,E1 8674.592,E2 8674.592} C_VEL
LIN {X 0,Y 587.315,Z 707.31,A -85,B 0,C 180,E1 8680.173,E2 8680.173} C_VEL
LIN {X 0,Y 587.308,Z 707.31,A -85,B 0,C 180,E1 8686.262,E2 8686.262} C_VEL
LIN {X 0,Y 587.306,Z 707.31,A -85,B 0,C 180,E1 8688.444,E2 8688.444} C_VEL
LIN {X 0,Y 592.581,Z 718.151,A -85,B 0,C 180,E1 8689.074,E2 8689.074} C_VEL
LIN {X 0,Y 612.74,Z 759.479,A -85,B 0,C 180,E1 8691.39,E2 8691.39} C_VEL
LIN {X 0,Y 615.126,Z 767.56,A -85,B 0,C 180,E1 8691.777,E2 8691.777} C_VEL
LIN {X 0,Y 611.953,Z 812.856,A -85,B 0,C 180,E1 8693.148,E2 8693.148} C_VEL
LIN {X 0,Y 607.704,Z 857.567,A -85,B 0,C 180,E1 8695.179,E2 8695.179} C_VEL
LIN {X 0,Y 603.21,Z 898.916,A -85,B 0,C 180,E1 8697.786,E2 8697.786} C_VEL
LIN {X 0,Y 598.473,Z 937.588,A -85,B 0,C 180,E1 8701.033,E2 8701.033} C_VEL
LIN {X 0,Y 594.425,Z 971.586,A -85,B 0,C 180,E1 8704.799,E2 8704.799} C_VEL
LIN {X 0,Y 591.466,Z 1000.172,A -85,B 0,C 180,E1 8708.981,E2 8708.981} C_VEL
LIN {X 0,Y 589.692,Z 1021.863,A -85,B 0,C 180,E1 8713.196,E2 8713.196} C_VEL
LIN {X 0,Y 588.845,Z 1037.366,A -85,B 0,C 180,E1 8717.366,E2 8717.366} C_VEL
LIN {X 0,Y 588.458,Z 1046.802,A -85,B 0,C 180,E1 8721.112,E2 8721.112} C_VEL
LIN {X 0,Y 588.334,Z 1052.608,A -85,B 0,C 180,E1 8725.569,E2 8725.569} C_VEL
LIN {X 0,Y 588.535,Z 1052.845,A -85,B 0,C 180,E1 8730.001,E2 8730.001} C_VEL
LIN {X 0,Y 588.476,Z 1047.537,A -85,B 0,C 180,E1 8734.431,E2 8734.431} C_VEL
LIN {X 0,Y 588.78,Z 1036.328,A -85,B 0,C 180,E1 8738.884,E2 8738.884} C_VEL
LIN {X 0,Y 589.761,Z 1020.19,A -85,B 0,C 180,E1 8743.079,E2 8743.079} C_VEL
LIN {X 0,Y 591.626,Z 997.758,A -85,B 0,C 180,E1 8747.324,E2 8747.324} C_VEL
LIN {X 0,Y 594.504,Z 970.557,A -85,B 0,C 180,E1 8751.24,E2 8751.24} C_VEL
LIN {X 0,Y 598.637,Z 936.381,A -85,B 0,C 180,E1 8754.988,E2 8754.988} C_VEL
LIN {X 0,Y 603.406,Z 897.369,A -85,B 0,C 180,E1 8758.23,E2 8758.23} C_VEL
LIN {X 0,Y 608.045,Z 855.684,A -85,B 0,C 180,E1 8760.825,E2 8760.825} C_VEL
LIN {X 0,Y 612.054,Z 812.589,A -85,B 0,C 180,E1 8762.756,E2 8762.756} C_VEL
LIN {X 0,Y 615.066,Z 768.813,A -85,B 0,C 180,E1 8764.083,E2 8764.083} C_VEL
LIN {X 0,Y 613.837,Z 762.178,A -85,B 0,C 180,E1 8764.351,E2 8764.351} C_VEL
LIN {X 0,Y 591.583,Z 716.943,A -85,B 0,C 180,E1 8766.819,E2 8766.819} C_VEL
LIN {X 0,Y 587.319,Z 707.31,A -85,B 0,C 180,E1 8767.327,E2 8767.327} C_VEL
LIN {X 0,Y 587.26,Z 707.31,A -85,B 0,C 180,E1 8772.139,E2 8772.139} C_VEL
LIN {X 0,Y 587.324,Z 707.31,A -85,B 0,C 180,E1 8777.865,E2 8777.865} C_VEL
LIN {X 0,Y 587.296,Z 707.31,A -85,B 0,C 180,E1 8783.594,E2 8783.594} C_VEL
LIN {X 0,Y 587.403,Z 707.31,A -85,B 0,C 180,E1 8788.935,E2 8788.935} C_VEL
LIN {X 0,Y 587.451,Z 707.31,A -85,B 0,C 180,E1 8794.539,E2 8794.539} C_VEL
LIN {X 0,Y 587.513,Z 707.31,A -85,B 0,C 180,E1 8800.406,E2 8800.406} C_VEL
LIN {X 0,Y 587.891,Z 707.31,A -85,B 0,C 180,E1 8806.583,E2 8806.583} C_VEL
LIN {X 0,Y 588.017,Z 707.31,A -85,B 0,C 180,E1 8812.594,E2 8812.594} C_VEL
LIN {X 0,Y 587.724,Z 707.31,A -85,B 0,C 180,E1 8817.041,E2 8817.041} C_VEL
LIN {X 0,Y 588.168,Z 707.31,A -85,B 0,C 180,E1 8821.474,E2 8821.474} C_VEL
LIN {X 0,Y 588.113,Z 707.31,A -85,B 0,C 180,E1 8827.4,E2 8827.4} C_VEL
LIN {X 0,Y 587.745,Z 707.31,A -85,B 0,C 180,E1 8833.415,E2 8833.415} C_VEL
LIN {X 0,Y 587.493,Z 707.31,A -85,B 0,C 180,E1 8839.589,E2 8839.589} C_VEL
LIN {X 0,Y 587.426,Z 707.31,A -85,B 0,C 180,E1 8845.456,E2 8845.456} C_VEL
LIN {X 0,Y 587.407,Z 707.31,A -85,B 0,C 180,E1 8851.058,E2 8851.058} C_VEL
LIN {X 0,Y 587.286,Z 707.31,A -85,B 0,C 180,E1 8856.878,E2 8856.878} C_VEL
LIN {X 0,Y 587.249,Z 707.31,A -85,B 0,C 180,E1 8862.135,E2 8862.135} C_VEL
LIN {X 0,Y 587.241,Z 707.31,A -85,B 0,C 180,E1 8867.859,E2 8867.859} C_VEL
LIN {X 0,Y 587.239,Z 707.31,A -85,B 0,C 180,E1 8870.247,E2 8870.247} C_VEL
LIN {X 0,Y 616.12,Z 765.907,A -85,B 0,C 180,E1 8873.276,E2 8873.276} C_VEL
LIN {X 0,Y 616.04,Z 770.795,A -85,B 0,C 180,E1 8873.355,E2 8873.355} C_VEL
LIN {X 0,Y 612.009,Z 787.874,A -85,B 0,C 180,E1 8873.452,E2 8873.452} C_VEL
LIN {X 0,Y 607.647,Z 804.71,A -85,B 0,C 180,E1 8873.64,E2 8873.64} C_VEL
LIN {X 0,Y 603.965,Z 852.102,A -85,B 0,C 180,E1 8875.247,E2 8875.247} C_VEL
LIN {X 0,Y 599.267,Z 897.188,A -85,B 0,C 180,E1 8877.495,E2 8877.495} C_VEL
LIN {X 0,Y 594.27,Z 939.516,A -85,B 0,C 180,E1 8880.406,E2 8880.406} C_VEL
LIN {X 0,Y 589.551,Z 977.557,A -85,B 0,C 180,E1 8883.884,E2 8883.884} C_VEL
LIN {X 0,Y 585.621,Z 1011.376,A -85,B 0,C 180,E1 8887.962,E2 8887.962} C_VEL
LIN {X 0,Y 582.962,Z 1038.078,A -85,B 0,C 180,E1 8892.215,E2 8892.215} C_VEL
LIN {X 0,Y 581.525,Z 1057.594,A -85,B 0,C 180,E1 8896.435,E2 8896.435} C_VEL
LIN {X 0,Y 580.894,Z 1070.23,A -85,B 0,C 180,E1 8900.237,E2 8900.237} C_VEL
LIN {X 0,Y 580.573,Z 1079.665,A -85,B 0,C 180,E1 8904.758,E2 8904.758} C_VEL
LIN {X 0,Y 580.443,Z 1083.164,A -85,B 0,C 180,E1 8908.503,E2 8908.503} C_VEL
LIN {X 0,Y 580.598,Z 1082.213,A -85,B 0,C 180,E1 8912.992,E2 8912.992} C_VEL
LIN {X 0,Y 580.617,Z 1075.635,A -85,B 0,C 180,E1 8917.498,E2 8917.498} C_VEL
LIN {X 0,Y 581.215,Z 1063.173,A -85,B 0,C 180,E1 8922.039,E2 8922.039} C_VEL
LIN {X 0,Y 582.424,Z 1045.479,A -85,B 0,C 180,E1 8926.343,E2 8926.343} C_VEL
LIN {X 0,Y 584.606,Z 1020.085,A -85,B 0,C 180,E1 8930.783,E2 8930.783} C_VEL
LIN {X 0,Y 588.182,Z 988.56,A -85,B 0,C 180,E1 8934.91,E2 8934.91} C_VEL
LIN {X 0,Y 592.725,Z 951.836,A -85,B 0,C 180,E1 8938.566,E2 8938.566} C_VEL
LIN {X 0,Y 597.74,Z 910.851,A -85,B 0,C 180,E1 8941.653,E2 8941.653} C_VEL
LIN {X 0,Y 602.56,Z 867.43,A -85,B 0,C 180,E1 8944.079,E2 8944.079} C_VEL
LIN {X 0,Y 606.6,Z 822.307,A -85,B 0,C 180,E1 8945.856,E2 8945.856} C_VEL
LIN {X 0,Y 609.366,Z 777.063,A -85,B 0,C 180,E1 8946.999,E2 8946.999} C_VEL
LIN {X 0,Y 609.071,Z 766.451,A -85,B 0,C 180,E1 8947.239,E2 8947.239} C_VEL
LIN {X 0,Y 586.309,Z 721.345,A -85,B 0,C 180,E1 8949.721,E2 8949.721} C_VEL
LIN {X 0,Y 579.467,Z 708.427,A -85,B 0,C 180,E1 8950.504,E2 8950.504} C_VEL
LIN {X 0,Y 579.373,Z 707.31,A -85,B 0,C 180,E1 8950.671,E2 8950.671} C_VEL
LIN {X 0,Y 579.296,Z 707.31,A -85,B 0,C 180,E1 8957.15,E2 8957.15} C_VEL
LIN {X 0,Y 579.362,Z 707.31,A -85,B 0,C 180,E1 8963.02,E2 8963.02} C_VEL
LIN {X 0,Y 579.523,Z 707.31,A -85,B 0,C 180,E1 8968.471,E2 8968.471} C_VEL
LIN {X 0,Y 579.5,Z 707.31,A -85,B 0,C 180,E1 8973.609,E2 8973.609} C_VEL
LIN {X 0,Y 579.502,Z 707.31,A -85,B 0,C 180,E1 8978.528,E2 8978.528} C_VEL
LIN {X 0,Y 579.733,Z 707.31,A -85,B 0,C 180,E1 8984.85,E2 8984.85} C_VEL
LIN {X 0,Y 580.04,Z 707.31,A -85,B 0,C 180,E1 8989.465,E2 8989.465} C_VEL
LIN {X 0,Y 579.974,Z 707.31,A -85,B 0,C 180,E1 8994.004,E2 8994.004} C_VEL
LIN {X 0,Y 580.083,Z 707.31,A -85,B 0,C 180,E1 9000.003,E2 9000.003} C_VEL
LIN {X 0,Y 579.891,Z 707.31,A -85,B 0,C 180,E1 9006.003,E2 9006.003} C_VEL
LIN {X 0,Y 579.913,Z 707.31,A -85,B 0,C 180,E1 9012.069,E2 9012.069} C_VEL
LIN {X 0,Y 579.593,Z 707.31,A -85,B 0,C 180,E1 9018.288,E2 9018.288} C_VEL
LIN {X 0,Y 579.564,Z 707.31,A -85,B 0,C 180,E1 9023.774,E2 9023.774} C_VEL
LIN {X 0,Y 579.333,Z 707.31,A -85,B 0,C 180,E1 9029.804,E2 9029.804} C_VEL
LIN {X 0,Y 579.292,Z 707.31,A -85,B 0,C 180,E1 9035.813,E2 9035.813} C_VEL
LIN {X 0,Y 579.399,Z 707.31,A -85,B 0,C 180,E1 9040.837,E2 9040.837} C_VEL
LIN {X 0,Y 579.34,Z 707.31,A -85,B 0,C 180,E1 9047.15,E2 9047.15} C_VEL
LIN {X 0,Y 579.388,Z 707.417,A -85,B 0,C 180,E1 9047.806,E2 9047.806} C_VEL
LIN {X 0,Y 584.401,Z 717.848,A -85,B 0,C 180,E1 9048.398,E2 9048.398} C_VEL
LIN {X 0,Y 604.54,Z 757.836,A -85,B 0,C 180,E1 9050.755,E2 9050.755} C_VEL
LIN {X 0,Y 608.671,Z 769.695,A -85,B 0,C 180,E1 9051.377,E2 9051.377} C_VEL
LIN {X 0,Y 605.395,Z 813.866,A -85,B 0,C 180,E1 9052.745,E2 9052.745} C_VEL
LIN {X 0,Y 600.945,Z 858.398,A -85,B 0,C 180,E1 9054.798,E2 9054.798} C_VEL
LIN {X 0,Y 596.215,Z 899.231,A -85,B 0,C 180,E1 9057.403,E2 9057.403} C_VEL
LIN {X 0,Y 591.355,Z 937.131,A -85,B 0,C 180,E1 9060.612,E2 9060.612} C_VEL
LIN {X 0,Y 586.959,Z 972.188,A -85,B 0,C 180,E1 9064.541,E2 9064.541} C_VEL
LIN {X 0,Y 583.861,Z 1000.221,A -85,B 0,C 180,E1 9068.694,E2 9068.694} C_VEL
LIN {X 0,Y 581.936,Z 1021.736,A -85,B 0,C 180,E1 9072.966,E2 9072.966} C_VEL
LIN {X 0,Y 580.981,Z 1037.278,A -85,B 0,C 180,E1 9077.191,E2 9077.191} C_VEL
LIN {X 0,Y 580.576,Z 1046.744,A -85,B 0,C 180,E1 9080.991,E2 9080.991} C_VEL
LIN {X 0,Y 580.427,Z 1052.589,A -85,B 0,C 180,E1 9085.508,E2 9085.508} C_VEL
LIN {X 0,Y 580.633,Z 1052.864,A -85,B 0,C 180,E1 9090.001,E2 9090.001} C_VEL
LIN {X 0,Y 580.578,Z 1047.582,A -85,B 0,C 180,E1 9094.492,E2 9094.492} C_VEL
LIN {X 0,Y 580.906,Z 1036.415,A -85,B 0,C 180,E1 9099.006,E2 9099.006} C_VEL
LIN {X 0,Y 581.958,Z 1020.173,A -85,B 0,C 180,E1 9103.297,E2 9103.297} C_VEL
LIN {X 0,Y 583.971,Z 998.151,A -85,B 0,C 180,E1 9107.558,E2 9107.558} C_VEL
LIN {X 0,Y 587.044,Z 970.831,A -85,B 0,C 180,E1 9111.546,E2 9111.546} C_VEL
LIN {X 0,Y 591.437,Z 936.899,A -85,B 0,C 180,E1 9115.314,E2 9115.314} C_VEL
LIN {X 0,Y 596.363,Z 898.641,A -85,B 0,C 180,E1 9118.543,E2 9118.543} C_VEL
LIN {X 0,Y 601.301,Z 856.119,A -85,B 0,C 180,E1 9121.224,E2 9121.224} C_VEL
LIN {X 0,Y 605.5,Z 812.852,A -85,B 0,C 180,E1 9123.179,E2 9123.179} C_VEL
LIN {X 0,Y 608.185,Z 766.972,A -85,B 0,C 180,E1 9124.607,E2 9124.607} C_VEL
LIN {X 0,Y 587.764,Z 724.38,A -85,B 0,C 180,E1 9127,E2 9127} C_VEL
LIN {X 0,Y 579.573,Z 709.015,A -85,B 0,C 180,E1 9127.888,E2 9127.888} C_VEL
LIN {X 0,Y 579.376,Z 707.31,A -85,B 0,C 180,E1 9128.027,E2 9128.027} C_VEL
LIN {X 0,Y 579.323,Z 707.31,A -85,B 0,C 180,E1 9132.907,E2 9132.907} C_VEL
LIN {X 0,Y 579.389,Z 707.31,A -85,B 0,C 180,E1 9139.333,E2 9139.333} C_VEL
LIN {X 0,Y 579.375,Z 707.31,A -85,B 0,C 180,E1 9144.868,E2 9144.868} C_VEL
LIN {X 0,Y 579.473,Z 707.31,A -85,B 0,C 180,E1 9150.204,E2 9150.204} C_VEL
LIN {X 0,Y 579.466,Z 707.31,A -85,B 0,C 180,E1 9156.251,E2 9156.251} C_VEL
LIN {X 0,Y 579.568,Z 707.31,A -85,B 0,C 180,E1 9161.711,E2 9161.711} C_VEL
LIN {X 0,Y 579.954,Z 707.31,A -85,B 0,C 180,E1 9166.396,E2 9166.396} C_VEL
LIN {X 0,Y 580.053,Z 707.31,A -85,B 0,C 180,E1 9171.83,E2 9171.83} C_VEL
LIN {X 0,Y 579.828,Z 707.31,A -85,B 0,C 180,E1 9177.001,E2 9177.001} C_VEL
LIN {X 0,Y 580.254,Z 707.31,A -85,B 0,C 180,E1 9181.494,E2 9181.494} C_VEL
LIN {X 0,Y 580.21,Z 707.31,A -85,B 0,C 180,E1 9187.501,E2 9187.501} C_VEL
LIN {X 0,Y 579.958,Z 707.31,A -85,B 0,C 180,E1 9192.063,E2 9192.063} C_VEL
LIN {X 0,Y 579.567,Z 707.31,A -85,B 0,C 180,E1 9198.283,E2 9198.283} C_VEL
LIN {X 0,Y 579.44,Z 707.31,A -85,B 0,C 180,E1 9203.743,E2 9203.743} C_VEL
LIN {X 0,Y 579.52,Z 707.31,A -85,B 0,C 180,E1 9208.075,E2 9208.075} C_VEL
LIN {X 0,Y 579.463,Z 707.31,A -85,B 0,C 180,E1 9213.308,E2 9213.308} C_VEL
LIN {X 0,Y 579.334,Z 707.31,A -85,B 0,C 180,E1 9218.883,E2 9218.883} C_VEL
LIN {X 0,Y 579.308,Z 707.31,A -85,B 0,C 180,E1 9225.065,E2 9225.065} C_VEL
LIN {X 0,Y 579.364,Z 707.31,A -85,B 0,C 180,E1 9229.637,E2 9229.637} C_VEL
LIN {X 0,Y 586.614,Z 722.283,A -85,B 0,C 180,E1 9230.46,E2 9230.46} C_VEL
LIN {X 0,Y 609.564,Z 768.28,A -85,B 0,C 180,E1 9232.868,E2 9232.868} C_VEL
LIN {X 0,Y 607.647,Z 804.71,A -85,B 0,C 180,E1 9233.64,E2 9233.64} C_VEL
LIN {X 0,Y 603.177,Z 821.522,A -85,B 0,C 180,E1 9233.911,E2 9233.911} C_VEL
LIN {X 0,Y 598.7,Z 837.933,A -85,B 0,C 180,E1 9234.27,E2 9234.27} C_VEL
LIN {X 0,Y 594.194,Z 881.856,A -85,B 0,C 180,E1 9236.231,E2 9236.231} C_VEL
LIN {X 0,Y 588.966,Z 925.317,A -85,B 0,C 180,E1 9238.945,E2 9238.945} C_VEL
LIN {X 0,Y 583.701,Z 965.722,A -85,B 0,C 180,E1 9242.349,E2 9242.349} C_VEL
LIN {X 0,Y 579.24,Z 1000.987,A -85,B 0,C 180,E1 9246.292,E2 9246.292} C_VEL
LIN {X 0,Y 575.899,Z 1030.127,A -85,B 0,C 180,E1 9250.588,E2 9250.588} C_VEL
LIN {X 0,Y 574.035,Z 1052.801,A -85,B 0,C 180,E1 9255.084,E2 9255.084} C_VEL
LIN {X 0,Y 573.044,Z 1069.158,A -85,B 0,C 180,E1 9259.717,E2 9259.717} C_VEL
LIN {X 0,Y 572.681,Z 1078.455,A -85,B 0,C 180,E1 9263.923,E2 9263.923} C_VEL
LIN {X 0,Y 572.542,Z 1083.164,A -85,B 0,C 180,E1 9268.483,E2 9268.483} C_VEL
LIN {X 0,Y 572.691,Z 1082.212,A -85,B 0,C 180,E1 9273.033,E2 9273.033} C_VEL
LIN {X 0,Y 572.719,Z 1075.635,A -85,B 0,C 180,E1 9277.602,E2 9277.602} C_VEL
LIN {X 0,Y 573.357,Z 1063.586,A -85,B 0,C 180,E1 9282.079,E2 9282.079} C_VEL
LIN {X 0,Y 574.607,Z 1045.076,A -85,B 0,C 180,E1 9286.608,E2 9286.608} C_VEL
LIN {X 0,Y 576.905,Z 1020.484,A -85,B 0,C 180,E1 9290.975,E2 9290.975} C_VEL
LIN {X 0,Y 580.724,Z 988.788,A -85,B 0,C 180,E1 9295.199,E2 9295.199} C_VEL
LIN {X 0,Y 585.576,Z 951.81,A -85,B 0,C 180,E1 9298.93,E2 9298.93} C_VEL
LIN {X 0,Y 590.847,Z 910.893,A -85,B 0,C 180,E1 9302.053,E2 9302.053} C_VEL
LIN {X 0,Y 595.915,Z 867.337,A -85,B 0,C 180,E1 9304.513,E2 9304.513} C_VEL
LIN {X 0,Y 600.267,Z 821.623,A -85,B 0,C 180,E1 9306.322,E2 9306.322} C_VEL
LIN {X 0,Y 603.202,Z 775.535,A -85,B 0,C 180,E1 9307.481,E2 9307.481} C_VEL
LIN {X 0,Y 602.354,Z 768.236,A -85,B 0,C 180,E1 9307.701,E2 9307.701} C_VEL
LIN {X 0,Y 579.88,Z 723.598,A -85,B 0,C 180,E1 9310.225,E2 9310.225} C_VEL
LIN {X 0,Y 571.585,Z 708.836,A -85,B 0,C 180,E1 9311.19,E2 9311.19} C_VEL
LIN {X 0,Y 571.409,Z 707.31,A -85,B 0,C 180,E1 9311.325,E2 9311.325} C_VEL
LIN {X 0,Y 571.341,Z 707.31,A -85,B 0,C 180,E1 9316.405,E2 9316.405} C_VEL
LIN {X 0,Y 571.434,Z 707.31,A -85,B 0,C 180,E1 9322.709,E2 9322.709} C_VEL
LIN {X 0,Y 571.571,Z 707.31,A -85,B 0,C 180,E1 9328.038,E2 9328.038} C_VEL
LIN {X 0,Y 571.607,Z 707.31,A -85,B 0,C 180,E1 9333.215,E2 9333.215} C_VEL
LIN {X 0,Y 571.558,Z 707.31,A -85,B 0,C 180,E1 9338.214,E2 9338.214} C_VEL
LIN {X 0,Y 571.691,Z 707.31,A -85,B 0,C 180,E1 9343.05,E2 9343.05} C_VEL
LIN {X 0,Y 572.035,Z 707.31,A -85,B 0,C 180,E1 9348.57,E2 9348.57} C_VEL
LIN {X 0,Y 572.097,Z 707.31,A -85,B 0,C 180,E1 9353.921,E2 9353.921} C_VEL
LIN {X 0,Y 572.179,Z 707.31,A -85,B 0,C 180,E1 9360.003,E2 9360.003} C_VEL
LIN {X 0,Y 571.971,Z 707.31,A -85,B 0,C 180,E1 9366.086,E2 9366.086} C_VEL
LIN {X 0,Y 571.989,Z 707.31,A -85,B 0,C 180,E1 9372.239,E2 9372.239} C_VEL
LIN {X 0,Y 571.694,Z 707.31,A -85,B 0,C 180,E1 9378.55,E2 9378.55} C_VEL
LIN {X 0,Y 571.711,Z 707.31,A -85,B 0,C 180,E1 9383.431,E2 9383.431} C_VEL
LIN {X 0,Y 571.385,Z 707.31,A -85,B 0,C 180,E1 9388.932,E2 9388.932} C_VEL
LIN {X 0,Y 571.384,Z 707.31,A -85,B 0,C 180,E1 9394.699,E2 9394.699} C_VEL
LIN {X 0,Y 571.39,Z 707.31,A -85,B 0,C 180,E1 9399.726,E2 9399.726} C_VEL
LIN {X 0,Y 571.373,Z 707.31,A -85,B 0,C 180,E1 9405.736,E2 9405.736} C_VEL
LIN {X 0,Y 571.459,Z 707.31,A -85,B 0,C 180,E1 9407.09,E2 9407.09} C_VEL
LIN {X 0,Y 575.957,Z 717.048,A -85,B 0,C 180,E1 9407.664,E2 9407.664} C_VEL
LIN {X 0,Y 596.544,Z 756.703,A -85,B 0,C 180,E1 9410.122,E2 9410.122} C_VEL
LIN {X 0,Y 602.258,Z 771.752,A -85,B 0,C 180,E1 9410.967,E2 9410.967} C_VEL
LIN {X 0,Y 598.863,Z 815.158,A -85,B 0,C 180,E1 9412.344,E2 9412.344} C_VEL
LIN {X 0,Y 594.297,Z 858.606,A -85,B 0,C 180,E1 9414.371,E2 9414.371} C_VEL
LIN {X 0,Y 589.219,Z 899.969,A -85,B 0,C 180,E1 9417.042,E2 9417.042} C_VEL
LIN {X 0,Y 584.066,Z 938.236,A -85,B 0,C 180,E1 9420.337,E2 9420.337} C_VEL
LIN {X 0,Y 579.605,Z 972.182,A -85,B 0,C 180,E1 9424.194,E2 9424.194} C_VEL
LIN {X 0,Y 576.275,Z 1000.265,A -85,B 0,C 180,E1 9428.399,E2 9428.399} C_VEL
LIN {X 0,Y 574.038,Z 1023.507,A -85,B 0,C 180,E1 9433.12,E2 9433.12} C_VEL
LIN {X 0,Y 573.033,Z 1039.502,A -85,B 0,C 180,E1 9437.787,E2 9437.787} C_VEL
LIN {X 0,Y 572.651,Z 1049.281,A -85,B 0,C 180,E1 9442.397,E2 9442.397} C_VEL
LIN {X 0,Y 572.464,Z 1053.284,A -85,B 0,C 180,E1 9446.966,E2 9446.966} C_VEL
LIN {X 0,Y 572.756,Z 1052.883,A -85,B 0,C 180,E1 9450.001,E2 9450.001} C_VEL
LIN {X 0,Y 572.688,Z 1047.626,A -85,B 0,C 180,E1 9454.554,E2 9454.554} C_VEL
LIN {X 0,Y 573.01,Z 1037.642,A -85,B 0,C 180,E1 9458.747,E2 9458.747} C_VEL
LIN {X 0,Y 574.035,Z 1022.777,A -85,B 0,C 180,E1 9462.967,E2 9462.967} C_VEL
LIN {X 0,Y 576.101,Z 1000.841,A -85,B 0,C 180,E1 9467.411,E2 9467.411} C_VEL
LIN {X 0,Y 579.516,Z 971.973,A -85,B 0,C 180,E1 9471.747,E2 9471.747} C_VEL
LIN {X 0,Y 584.092,Z 938.375,A -85,B 0,C 180,E1 9475.553,E2 9475.553} C_VEL
LIN {X 0,Y 589.346,Z 899.526,A -85,B 0,C 180,E1 9478.888,E2 9478.888} C_VEL
LIN {X 0,Y 594.585,Z 856.712,A -85,B 0,C 180,E1 9481.618,E2 9481.618} C_VEL
LIN {X 0,Y 598.864,Z 814.301,A -85,B 0,C 180,E1 9483.564,E2 9483.564} C_VEL
LIN {X 0,Y 601.481,Z 769.301,A -85,B 0,C 180,E1 9485.014,E2 9485.014} C_VEL
